C05370=1019.467,-110.317,-113.060,-23.964,21.692,-44.427
C05371=1019.463,-110.709,-113.032,-23.963,21.693,-44.433
C05372=1019.458,-111.102,-113.004,-23.963,21.694,-44.439
C05373=1019.453,-111.495,-112.976,-23.962,21.694,-44.446
C05374=1019.448,-111.888,-112.949,-23.961,21.694,-44.451
C05375=1019.443,-112.281,-112.921,-23.960,21.695,-44.456
C05376=1019.437,-112.673,-112.893,-23.959,21.696,-44.462
C05377=1019.433,-113.065,-112.866,-23.959,21.696,-44.468
C05378=1019.428,-113.458,-112.838,-23.958,21.697,-44.473
C05379=1019.423,-113.850,-112.811,-23.957,21.698,-44.479
C05380=1019.418,-114.243,-112.783,-23.957,21.699,-44.485
C05381=1019.412,-114.635,-112.756,-23.956,21.700,-44.490
C05382=1019.407,-115.028,-112.728,-23.955,21.701,-44.496
C05383=1019.402,-115.420,-112.701,-23.954,21.700,-44.501
C05384=1019.397,-115.813,-112.673,-23.954,21.701,-44.507
C05385=1019.392,-116.205,-112.645,-23.953,21.702,-44.512
C05386=1019.387,-116.598,-112.617,-23.952,21.703,-44.518
C05387=1019.381,-116.990,-112.590,-23.952,21.704,-44.523
C05388=1019.376,-117.382,-112.562,-23.951,21.705,-44.529
C05389=1019.370,-117.774,-112.535,-23.950,21.705,-44.536
C05390=1019.365,-118.167,-112.507,-23.949,21.705,-44.541
C05391=1019.360,-118.558,-112.480,-23.948,21.706,-44.547
C05392=1019.354,-118.951,-112.452,-23.948,21.706,-44.553
C05393=1019.349,-119.343,-112.425,-23.947,21.707,-44.558
C05394=1019.343,-119.736,-112.398,-23.946,21.708,-44.564
C05395=1019.338,-120.127,-112.370,-23.946,21.709,-44.569
C05396=1019.332,-120.520,-112.343,-23.945,21.710,-44.575
C05397=1019.327,-120.912,-112.315,-23.944,21.710,-44.580
C05398=1019.321,-121.304,-112.288,-23.943,21.710,-44.586
C05399=1019.315,-121.696,-112.260,-23.943,21.711,-44.591
C05400=1019.310,-122.088,-112.233,-23.942,21.712,-44.597
C05401=1019.304,-122.480,-112.206,-23.941,21.713,-44.603
C05402=1019.299,-122.872,-112.179,-23.941,21.714,-44.608
C05403=1019.292,-123.264,-112.151,-23.940,21.715,-44.614
C05404=1019.287,-123.656,-112.124,-23.939,21.714,-44.619
C05405=1019.281,-124.049,-112.097,-23.939,21.715,-44.625
C05406=1019.275,-124.440,-112.070,-23.938,21.716,-44.630
C05407=1019.269,-124.832,-112.042,-23.937,21.717,-44.636
C05408=1019.264,-125.224,-112.015,-23.936,21.718,-44.642
C05409=1019.257,-125.616,-111.988,-23.936,21.719,-44.647
C05410=1019.252,-126.008,-111.961,-23.935,21.719,-44.652
C05411=1019.246,-126.399,-111.934,-23.934,21.719,-44.658
C05412=1019.240,-126.792,-111.906,-23.934,21.720,-44.664
C05413=1019.234,-127.183,-111.880,-23.933,21.721,-44.669
C05414=1019.228,-127.576,-111.852,-23.932,21.722,-44.675
C05415=1019.222,-127.967,-111.825,-23.932,21.723,-44.680
C05416=1019.216,-128.359,-111.798,-23.931,21.723,-44.686
C05417=1019.210,-128.751,-111.771,-23.930,21.723,-44.691
C05418=1019.203,-129.143,-111.744,-23.929,21.724,-44.697
C05419=1019.198,-129.534,-111.717,-23.929,21.725,-44.703
C05420=1019.191,-129.927,-111.690,-23.928,21.726,-44.708
C05421=1019.185,-130.318,-111.663,-23.927,21.727,-44.714
C05422=1019.179,-130.711,-111.636,-23.926,21.727,-44.719
C05423=1019.173,-131.102,-111.609,-23.926,21.728,-44.725
C05424=1019.167,-131.493,-111.582,-23.925,21.728,-44.730
C05425=1019.160,-131.886,-111.555,-23.924,21.729,-44.736
C05426=1019.154,-132.277,-111.528,-23.924,21.730,-44.741
C05427=1019.148,-132.669,-111.501,-23.923,21.730,-44.747
C05428=1019.141,-133.061,-111.474,-23.922,21.731,-44.752
C05429=1019.135,-133.452,-111.448,-23.922,21.732,-44.758
C05430=1019.128,-133.844,-111.420,-23.921,21.732,-44.763
C05431=1019.504,-133.817,-111.655,-23.921,21.732,-44.763
C05432=1019.511,-133.425,-111.682,-23.922,21.732,-44.758
C05433=1019.517,-133.034,-111.709,-23.922,21.731,-44.752
C05434=1019.524,-132.641,-111.736,-23.923,21.730,-44.747
C05435=1019.530,-132.250,-111.762,-23.924,21.730,-44.741
C05436=1019.537,-131.858,-111.790,-23.924,21.729,-44.736
C05437=1019.542,-131.466,-111.816,-23.925,21.728,-44.730
C05438=1019.548,-131.075,-111.843,-23.926,21.728,-44.725
C05439=1019.554,-130.683,-111.871,-23.926,21.727,-44.719
C05440=1019.560,-130.291,-111.897,-23.927,21.727,-44.714
C05441=1019.567,-129.899,-111.924,-23.928,21.726,-44.708
C05442=1019.573,-129.508,-111.951,-23.929,21.725,-44.703
C05443=1019.578,-129.116,-111.978,-23.929,21.724,-44.697
C05444=1019.585,-128.723,-112.005,-23.930,21.723,-44.691
C05445=1019.591,-128.332,-112.032,-23.931,21.723,-44.686
C05446=1019.596,-127.940,-112.059,-23.932,21.723,-44.680
C05447=1019.603,-127.548,-112.086,-23.932,21.722,-44.675
C05448=1019.609,-127.157,-112.113,-23.933,21.721,-44.669
C05449=1019.615,-126.764,-112.141,-23.934,21.720,-44.664
C05450=1019.621,-126.373,-112.167,-23.934,21.719,-44.658
C05451=1019.626,-125.981,-112.194,-23.935,21.719,-44.652
C05452=1019.633,-125.589,-112.222,-23.936,21.719,-44.647
C05453=1019.638,-125.197,-112.249,-23.936,21.718,-44.642
C05454=1019.643,-124.805,-112.276,-23.937,21.717,-44.636
C05455=1019.650,-124.413,-112.303,-23.938,21.716,-44.630
C05456=1019.655,-124.021,-112.330,-23.939,21.715,-44.625
C05457=1019.661,-123.629,-112.357,-23.939,21.714,-44.619
C05458=1019.666,-123.237,-112.385,-23.940,21.715,-44.614
C05459=1019.672,-122.845,-112.411,-23.941,21.714,-44.608
C05460=1019.678,-122.453,-112.439,-23.941,21.713,-44.603
C05461=1019.684,-122.061,-112.466,-23.942,21.712,-44.597
C05462=1019.689,-121.669,-112.493,-23.943,21.711,-44.591
C05463=1019.695,-121.277,-112.521,-23.943,21.710,-44.586
C05464=1019.700,-120.885,-112.548,-23.944,21.710,-44.580
C05465=1019.705,-120.493,-112.576,-23.945,21.710,-44.575
C05466=1019.711,-120.101,-112.603,-23.946,21.709,-44.569
C05467=1019.716,-119.709,-112.630,-23.946,21.708,-44.564
C05468=1019.722,-119.316,-112.657,-23.947,21.707,-44.558
C05469=1019.727,-118.924,-112.684,-23.948,21.706,-44.553
C05470=1019.732,-118.532,-112.712,-23.948,21.706,-44.547
C05471=1019.738,-118.140,-112.740,-23.949,21.705,-44.541
C05472=1019.743,-117.748,-112.767,-23.950,21.705,-44.536
C05473=1019.749,-117.355,-112.795,-23.951,21.705,-44.529
C05474=1019.754,-116.963,-112.822,-23.952,21.704,-44.523
C05475=1019.759,-116.570,-112.850,-23.952,21.703,-44.518
C05476=1019.764,-116.178,-112.877,-23.953,21.702,-44.512
C05477=1019.769,-115.786,-112.904,-23.954,21.701,-44.507
C05478=1019.774,-115.393,-112.932,-23.954,21.700,-44.501
C05479=1019.779,-115.001,-112.959,-23.955,21.701,-44.496
C05480=1019.785,-114.608,-112.987,-23.956,21.700,-44.490
C05481=1019.789,-114.216,-113.014,-23.957,21.699,-44.485
C05482=1019.795,-113.823,-113.042,-23.957,21.698,-44.479
C05483=1019.800,-113.432,-113.070,-23.958,21.697,-44.473
C05484=1019.805,-113.039,-113.098,-23.959,21.696,-44.468
C05485=1019.810,-112.647,-113.125,-23.959,21.696,-44.462
C05486=1019.815,-112.254,-113.153,-23.960,21.695,-44.456
C05487=1019.819,-111.862,-113.181,-23.961,21.694,-44.451
C05488=1019.825,-111.469,-113.209,-23.962,21.694,-44.446
C05489=1019.829,-111.076,-113.236,-23.963,21.694,-44.439
C05490=1019.834,-110.683,-113.263,-23.963,21.693,-44.433
C05491=1019.839,-110.290,-113.291,-23.964,21.692,-44.427
C05492=1019.844,-109.898,-113.319,-23.965,21.691,-44.422
C05493=1019.849,-109.505,-113.347,-23.965,21.691,-44.416
C05494=1019.854,-109.112,-113.375,-23.966,21.690,-44.411
C05495=1019.858,-108.719,-113.403,-23.967,21.689,-44.405
C05496=1019.863,-108.326,-113.431,-23.968,21.688,-44.399
C05497=1019.867,-107.934,-113.459,-23.968,21.688,-44.394
C05498=1019.872,-107.541,-113.487,-23.969,21.687,-44.388
C05499=1019.877,-107.147,-113.514,-23.970,21.687,-44.383
C05500=1019.881,-106.754,-113.543,-23.971,21.686,-44.376
C05501=1019.886,-106.362,-113.570,-23.971,21.686,-44.370
C05502=1019.891,-105.969,-113.598,-23.972,21.685,-44.365
C05503=1019.895,-105.576,-113.627,-23.973,21.684,-44.359
C05504=1019.900,-105.183,-113.655,-23.974,21.683,-44.353
C05505=1019.904,-104.791,-113.682,-23.974,21.682,-44.348
C05506=1019.909,-104.399,-113.710,-23.975,21.681,-44.342
C05507=1019.913,-104.008,-113.738,-23.976,21.682,-44.337
C05508=1019.918,-103.616,-113.766,-23.976,21.681,-44.331
C05509=1019.921,-103.227,-113.794,-23.977,21.680,-44.326
C05510=1019.926,-102.836,-113.822,-23.978,21.679,-44.320
C05511=1019.930,-102.447,-113.849,-23.979,21.678,-44.314
C05512=1019.935,-102.059,-113.878,-23.980,21.678,-44.307
C05513=1019.939,-101.672,-113.905,-23.980,21.677,-44.302
C05514=1019.943,-101.284,-113.933,-23.981,21.676,-44.296
C05515=1019.947,-100.898,-113.961,-23.982,21.677,-44.291
C05516=1019.952,-100.513,-113.988,-23.982,21.676,-44.285
C05517=1019.956,-100.127,-114.016,-23.983,21.675,-44.280
C05518=1019.960,-99.743,-114.044,-23.984,21.674,-44.274
C05519=1019.964,-99.358,-114.072,-23.985,21.673,-44.268
C05520=1019.968,-98.975,-114.099,-23.985,21.673,-44.263
C05521=1019.972,-98.591,-114.127,-23.986,21.673,-44.258
C05522=1019.976,-98.208,-114.154,-23.987,21.672,-44.252
C05523=1019.980,-97.825,-114.182,-23.988,21.671,-44.246
C05524=1019.984,-97.442,-114.209,-23.988,21.670,-44.241
C05525=1019.988,-97.058,-114.238,-23.989,21.669,-44.235
C05526=1019.991,-96.675,-114.265,-23.990,21.669,-44.230
C05527=1019.996,-96.291,-114.293,-23.990,21.668,-44.224
C05528=1020.000,-95.907,-114.321,-23.991,21.668,-44.219
C05529=1020.004,-95.522,-114.348,-23.992,21.667,-44.213
C05530=1020.007,-95.138,-114.376,-23.993,21.666,-44.207
C05531=1020.011,-94.752,-114.404,-23.994,21.666,-44.200
C05532=1020.015,-94.365,-114.432,-23.994,21.665,-44.195
C05533=1020.019,-93.979,-114.461,-23.995,21.664,-44.189
C05534=1020.023,-93.592,-114.489,-23.996,21.664,-44.184
C05535=1020.026,-93.203,-114.516,-23.996,21.664,-44.178
C05536=1020.027,-93.059,-114.527,-23.997,21.663,-44.176
C05537=1019.643,111.857,-131.928,-24.335,21.425,-41.686
C05538=1019.639,112.243,-131.965,-24.335,21.423,-41.684
C05539=1019.635,112.628,-132.001,-24.335,21.424,-41.681
C05540=1019.630,113.026,-132.039,-24.336,21.423,-41.677
C05541=1019.625,113.425,-132.077,-24.336,21.423,-41.675
C05542=1019.620,113.823,-132.115,-24.337,21.423,-41.671
C05543=1019.616,114.222,-132.152,-24.337,21.422,-41.668
C05544=1019.611,114.620,-132.190,-24.338,21.423,-41.664
C05545=1019.606,115.019,-132.228,-24.338,21.422,-41.662
C05546=1019.602,115.418,-132.266,-24.339,21.422,-41.659
C05547=1019.597,115.816,-132.304,-24.339,21.422,-41.655
C05548=1019.592,116.214,-132.341,-24.340,21.422,-41.652
C05549=1019.588,116.613,-132.380,-24.340,21.421,-41.649
C05550=1019.583,117.012,-132.417,-24.340,21.420,-41.646
C05551=1019.578,117.410,-132.455,-24.341,21.421,-41.642
C05552=1019.573,117.809,-132.493,-24.341,21.420,-41.638
C05553=1019.568,118.207,-132.531,-24.342,21.420,-41.637
C05554=1019.563,118.606,-132.569,-24.342,21.420,-41.633
C05555=1019.559,119.004,-132.607,-24.343,21.420,-41.629
C05556=1019.553,119.403,-132.644,-24.343,21.420,-41.626
C05557=1019.549,119.801,-132.683,-24.343,21.419,-41.624
C05558=1019.544,120.200,-132.721,-24.344,21.419,-41.620
C05559=1019.539,120.599,-132.759,-24.345,21.419,-41.617
C05560=1019.534,120.997,-132.797,-24.345,21.418,-41.614
C05561=1019.530,121.395,-132.835,-24.345,21.418,-41.611
C05562=1019.525,121.794,-132.873,-24.346,21.418,-41.607
C05563=1019.521,122.192,-132.912,-24.346,21.417,-41.605
C05564=1019.516,122.591,-132.949,-24.347,21.418,-41.602
C05565=1019.511,122.990,-132.988,-24.347,21.417,-41.598
C05566=1019.507,123.388,-133.026,-24.348,21.418,-41.595
C05567=1019.502,123.787,-133.064,-24.348,21.416,-41.592
C05568=1019.498,124.185,-133.103,-24.348,21.417,-41.589
C05569=1019.492,124.584,-133.140,-24.349,21.416,-41.585
C05570=1019.488,124.982,-133.179,-24.349,21.416,-41.583
C05571=1019.483,125.381,-133.217,-24.350,21.416,-41.580
C05572=1019.479,125.779,-133.255,-24.350,21.416,-41.576
C05573=1019.474,126.178,-133.294,-24.350,21.415,-41.574
C05574=1019.469,126.577,-133.332,-24.351,21.415,-41.571
C05575=1019.464,126.976,-133.370,-24.351,21.415,-41.567
C05576=1019.459,127.374,-133.409,-24.352,21.415,-41.565
C05577=1019.454,127.772,-133.447,-24.352,21.414,-41.561
C05578=1019.450,128.171,-133.485,-24.353,21.415,-41.558
C05579=1019.444,128.570,-133.523,-24.353,21.414,-41.555
C05580=1019.440,128.969,-133.562,-24.354,21.414,-41.552
C05581=1019.435,129.367,-133.600,-24.354,21.413,-41.550
C05582=1019.431,129.766,-133.638,-24.354,21.413,-41.547
C05583=1019.425,130.164,-133.677,-24.355,21.413,-41.543
C05584=1019.421,130.564,-133.715,-24.355,21.413,-41.541
C05585=1019.415,130.961,-133.753,-24.356,21.413,-41.538
C05586=1019.410,131.360,-133.792,-24.356,21.413,-41.534
C05587=1019.406,131.759,-133.830,-24.356,21.412,-41.532
C05588=1019.400,132.158,-133.869,-24.357,21.412,-41.528
C05589=1019.396,132.557,-133.907,-24.357,21.412,-41.525
C05590=1019.390,132.956,-133.946,-24.358,21.411,-41.523
C05591=1019.386,133.354,-133.984,-24.358,21.412,-41.519
C05592=1019.380,133.752,-134.023,-24.358,21.411,-41.517
C05593=1019.375,134.151,-134.061,-24.359,21.411,-41.514
C05594=1019.370,134.550,-134.100,-24.359,21.411,-41.510
C05595=1019.365,134.949,-134.138,-24.360,21.410,-41.508
C05596=1019.360,135.347,-134.177,-24.360,21.411,-41.505
C05597=1019.355,135.743,-134.214,-24.360,21.410,-41.502
C05598=1019.350,136.115,-134.250,-24.361,21.409,-41.500
C05599=1019.346,136.454,-134.283,-24.361,21.410,-41.497
C05600=1019.342,136.772,-134.314,-24.361,21.409,-41.495
C05601=1019.338,137.088,-134.345,-24.362,21.409,-41.491
C05602=1019.334,137.424,-134.377,-24.363,21.410,-41.488
C05603=1019.329,137.794,-134.413,-24.363,21.408,-41.486
C05604=1019.323,138.196,-134.452,-24.363,21.408,-41.484
C05605=1019.320,138.402,-134.471,-24.363,21.408,-41.482
C05606=1019.317,138.618,-134.492,-24.364,21.408,-41.480
C05607=1019.315,138.855,-134.515,-24.364,21.408,-41.478
C05608=1019.311,139.115,-134.541,-24.364,21.407,-41.476
C05609=1019.307,139.393,-134.567,-24.364,21.408,-41.475
C05610=1019.304,139.681,-134.596,-24.365,21.408,-41.473
C05611=1019.300,139.969,-134.623,-24.365,21.408,-41.471
C05612=1019.296,140.246,-134.650,-24.365,21.408,-41.470
C05613=1019.293,140.504,-134.675,-24.366,21.408,-41.468
C05614=1019.290,140.740,-134.697,-24.366,21.408,-41.466
C05615=1019.284,141.158,-134.738,-24.366,21.407,-41.462
C05616=1019.279,141.562,-134.777,-24.366,21.406,-41.460
C05617=1019.273,141.968,-134.817,-24.367,21.407,-41.457
C05618=1019.268,142.374,-134.855,-24.368,21.406,-41.453
C05619=1019.263,142.781,-134.895,-24.368,21.406,-41.451
C05620=1019.257,143.189,-134.935,-24.368,21.406,-41.448
C05621=1019.252,143.598,-134.974,-24.369,21.405,-41.445
C05622=1019.246,144.007,-135.014,-24.369,21.406,-41.442
C05623=1019.240,144.418,-135.054,-24.370,21.405,-41.438
C05624=1019.235,144.828,-135.093,-24.370,21.405,-41.436
C05625=1019.229,145.241,-135.133,-24.370,21.405,-41.432
C05626=1019.224,145.652,-135.173,-24.371,21.404,-41.431
C05627=1019.218,146.065,-135.214,-24.371,21.405,-41.427
C05628=1019.212,146.477,-135.254,-24.372,21.404,-41.424
C05629=1019.207,146.891,-135.293,-24.372,21.404,-41.422
C05630=1019.201,147.304,-135.334,-24.372,21.404,-41.418
C05631=1019.195,147.718,-135.374,-24.373,21.403,-41.416
C05632=1019.189,148.133,-135.414,-24.373,21.403,-41.412
C05633=1019.183,148.546,-135.455,-24.374,21.403,-41.409
C05634=1019.178,148.960,-135.495,-24.374,21.403,-41.407
C05635=1019.172,149.375,-135.535,-24.375,21.403,-41.403
C05636=1019.166,149.789,-135.575,-24.375,21.402,-41.401
C05637=1019.161,150.203,-135.615,-24.375,21.402,-41.398
C05638=1019.155,150.617,-135.655,-24.376,21.402,-41.394
C05639=1019.149,151.030,-135.695,-24.376,21.401,-41.392
C05640=1019.143,151.444,-135.736,-24.377,21.402,-41.389
C05641=1019.137,151.857,-135.776,-24.377,21.402,-41.387
C05642=1019.131,152.271,-135.816,-24.377,21.401,-41.383
C05643=1019.125,152.683,-135.856,-24.378,21.401,-41.381
C05644=1019.118,153.096,-135.896,-24.378,21.400,-41.377
C05645=1019.113,153.507,-135.936,-24.378,21.400,-41.375
C05646=1019.107,153.918,-135.977,-24.379,21.401,-41.372
C05647=1019.101,154.329,-136.017,-24.380,21.400,-41.368
C05648=1019.095,154.739,-136.056,-24.380,21.400,-41.366
C05649=1019.089,155.149,-136.096,-24.380,21.400,-41.363
C05650=1019.083,155.557,-136.136,-24.381,21.399,-41.361
C05651=1019.077,155.965,-136.176,-24.381,21.400,-41.358
C05652=1019.071,156.371,-136.215,-24.381,21.399,-41.355
C05653=1019.065,156.777,-136.255,-24.382,21.399,-41.352
C05654=1019.059,157.182,-136.294,-24.382,21.399,-41.350
C05655=1019.053,157.587,-136.334,-24.383,21.398,-41.346
C05656=1019.047,157.990,-136.373,-24.383,21.398,-41.344
C05657=1019.041,158.392,-136.413,-24.383,21.399,-41.341
C05658=1019.036,158.794,-136.452,-24.384,21.397,-41.339
C05659=1019.029,159.196,-136.491,-24.384,21.398,-41.335
C05660=1019.024,159.597,-136.530,-24.384,21.398,-41.333
C05661=1019.023,159.997,-136.573,-24.385,21.397,-41.330
C05662=1019.021,160.393,-136.614,-24.385,21.397,-41.328
C05663=1019.020,160.798,-136.656,-24.386,21.397,-41.325
C05664=1019.020,161.012,-136.679,-24.386,21.397,-41.324
C05665=1019.018,161.237,-136.702,-24.386,21.396,-41.322
C05666=1019.018,161.474,-136.727,-24.386,21.396,-41.320
C05667=1019.016,161.725,-136.753,-24.387,21.397,-41.319
C05668=1019.016,161.988,-136.781,-24.387,21.397,-41.317
C05669=1019.015,162.256,-136.809,-24.387,21.396,-41.315
C05670=1019.015,162.529,-136.837,-24.387,21.396,-41.313
C05671=1019.013,162.797,-136.866,-24.388,21.396,-41.311
C05672=1019.012,163.060,-136.893,-24.388,21.396,-41.309
C05673=1019.011,163.314,-136.920,-24.388,21.395,-41.308
C05674=1019.011,163.549,-136.945,-24.388,21.396,-41.306
C05675=1019.010,163.961,-136.989,-24.389,21.395,-41.304
C05676=1019.009,164.152,-137.008,-24.389,21.395,-41.302
C05677=1019.008,164.537,-137.049,-24.389,21.395,-41.300
C05678=1019.006,164.937,-137.091,-24.390,21.395,-41.297
C05679=1019.005,165.338,-137.133,-24.390,21.395,-41.295
C05680=1019.004,165.738,-137.176,-24.390,21.394,-41.291
C05681=1019.002,166.139,-137.217,-24.391,21.394,-41.289
C05682=1019.002,166.539,-137.259,-24.391,21.395,-41.286
C05683=1019.000,166.940,-137.302,-24.391,21.393,-41.284
C05684=1018.999,167.339,-137.344,-24.392,21.394,-41.280
C05685=1018.997,167.740,-137.387,-24.392,21.394,-41.278
C05686=1018.996,168.141,-137.428,-24.393,21.394,-41.275
C05687=1018.995,168.541,-137.471,-24.393,21.393,-41.273
C05688=1018.993,168.942,-137.513,-24.393,21.393,-41.271
C05689=1018.992,169.342,-137.555,-24.394,21.393,-41.267
C05690=1018.991,169.742,-137.598,-24.394,21.392,-41.265
C05691=1018.990,170.143,-137.640,-24.395,21.392,-41.262
C05692=1018.989,170.544,-137.683,-24.395,21.392,-41.260
C05693=1018.987,170.944,-137.726,-24.395,21.392,-41.256
C05694=1018.986,171.345,-137.768,-24.396,21.392,-41.254
C05695=1018.985,171.745,-137.811,-24.396,21.392,-41.251
C05696=1018.984,172.146,-137.853,-24.396,21.392,-41.249
C05697=1018.983,172.547,-137.895,-24.397,21.391,-41.247
C05698=1018.981,172.947,-137.938,-24.397,21.391,-41.243
C05699=1018.981,173.347,-137.980,-24.397,21.391,-41.242
C05700=1018.979,173.749,-138.023,-24.398,21.390,-41.238
C05701=1018.978,174.149,-138.066,-24.398,21.390,-41.236
C05702=1018.976,174.550,-138.109,-24.399,21.391,-41.233
C05703=1018.975,174.950,-138.150,-24.399,21.390,-41.231
C05704=1018.975,175.352,-138.193,-24.400,21.390,-41.227
C05705=1018.973,175.752,-138.236,-24.400,21.390,-41.225
C05706=1018.972,176.153,-138.279,-24.400,21.390,-41.223
C05707=1018.971,176.553,-138.321,-24.401,21.389,-41.219
C05708=1018.970,176.954,-138.364,-24.401,21.389,-41.218
C05709=1018.969,177.355,-138.407,-24.401,21.389,-41.214
C05710=1018.968,177.756,-138.450,-24.402,21.389,-41.212
C05711=1018.966,178.156,-138.493,-24.402,21.389,-41.209
C05712=1018.966,178.558,-138.535,-24.402,21.388,-41.207
C05713=1018.965,178.958,-138.578,-24.403,21.388,-41.205
C05714=1018.963,179.359,-138.621,-24.403,21.388,-41.201
C05715=1018.963,179.760,-138.664,-24.403,21.388,-41.199
C05716=1018.961,180.160,-138.707,-24.404,21.388,-41.196
C05717=1018.960,180.562,-138.751,-24.404,21.388,-41.194
C05718=1018.959,180.963,-138.793,-24.405,21.387,-41.190
C05719=1018.957,181.363,-138.836,-24.405,21.387,-41.188
C05720=1018.957,181.764,-138.879,-24.405,21.387,-41.186
C05721=1018.957,182.165,-138.922,-24.406,21.387,-41.183
C05722=1018.955,182.566,-138.965,-24.406,21.386,-41.181
C05723=1018.955,182.967,-139.008,-24.407,21.387,-41.177
C05724=1018.953,183.368,-139.051,-24.407,21.386,-41.176
C05725=1018.952,183.769,-139.094,-24.407,21.386,-41.172
C05726=1018.951,184.169,-139.137,-24.408,21.386,-41.170
C05727=1018.950,184.571,-139.181,-24.408,21.386,-41.168
C05728=1018.950,184.972,-139.224,-24.409,21.386,-41.165
C05729=1018.948,185.372,-139.267,-24.409,21.385,-41.162
C05730=1018.948,185.773,-139.310,-24.409,21.385,-41.159
C05731=1018.947,186.175,-139.354,-24.410,21.385,-41.157
C05732=1018.945,186.575,-139.397,-24.410,21.384,-41.155
C05733=1018.945,186.976,-139.440,-24.410,21.384,-41.151
C05734=1018.944,187.378,-139.483,-24.411,21.384,-41.150
C05735=1018.943,187.779,-139.526,-24.411,21.385,-41.146
C05736=1018.942,188.179,-139.569,-24.411,21.384,-41.144
C05737=1018.941,188.581,-139.613,-24.412,21.384,-41.141
C05738=1018.940,188.982,-139.656,-24.412,21.384,-41.139
C05739=1018.940,189.383,-139.699,-24.412,21.384,-41.137
C05740=1018.939,189.784,-139.743,-24.413,21.383,-41.133
C05741=1018.938,190.185,-139.787,-24.413,21.383,-41.131
C05742=1018.937,190.586,-139.831,-24.414,21.383,-41.128
C05743=1018.936,190.988,-139.874,-24.414,21.383,-41.126
C05744=1018.935,191.389,-139.917,-24.414,21.382,-41.124
C05745=1018.935,191.790,-139.961,-24.415,21.382,-41.120
C05746=1018.934,192.191,-140.005,-24.415,21.382,-41.118
C05747=1018.933,192.592,-140.048,-24.415,21.382,-41.115
C05748=1018.932,192.992,-140.091,-24.416,21.382,-41.113
C05749=1018.931,193.395,-140.135,-24.416,21.382,-41.109
C05750=1018.931,193.795,-140.179,-24.417,21.382,-41.108
C05751=1018.930,194.196,-140.222,-24.417,21.381,-41.105
C05752=1018.929,194.598,-140.266,-24.417,21.381,-41.102
C05753=1018.929,194.998,-140.310,-24.418,21.381,-41.100
C05754=1018.928,195.399,-140.353,-24.418,21.381,-41.097
C05755=1018.927,195.801,-140.397,-24.418,21.380,-41.094
C05756=1018.926,196.201,-140.441,-24.419,21.381,-41.091
C05757=1018.926,196.603,-140.485,-24.419,21.380,-41.089
C05758=1018.926,197.004,-140.529,-24.419,21.380,-41.087
C05759=1018.925,197.405,-140.572,-24.420,21.380,-41.084
C05760=1018.923,197.807,-140.616,-24.420,21.380,-41.082
C05761=1018.923,198.207,-140.660,-24.421,21.380,-41.078
C05762=1018.923,198.609,-140.704,-24.421,21.379,-41.076
C05763=1018.922,199.010,-140.748,-24.421,21.379,-41.074
C05764=1018.922,199.408,-140.791,-24.422,21.379,-41.071
C05765=1018.921,199.797,-140.834,-24.422,21.379,-41.069
C05766=1018.920,200.198,-140.878,-24.423,21.378,-41.065
C05767=1018.920,200.411,-140.901,-24.423,21.378,-41.065
C05768=1018.920,200.633,-140.926,-24.423,21.378,-41.063
C05769=1018.920,200.863,-140.951,-24.423,21.378,-41.061
C05770=1018.919,201.090,-140.976,-24.423,21.379,-41.060
C05771=1018.919,201.497,-141.020,-24.424,21.378,-41.058
C05772=1018.919,201.848,-141.059,-24.424,21.378,-41.054
C05773=1018.920,202.198,-141.099,-24.424,21.378,-41.052
C05774=1018.920,202.585,-141.142,-24.425,21.378,-41.051
C05775=1018.927,203.801,-141.279,-24.373,21.403,-41.416
C05776=1018.929,204.050,-141.306,-24.373,21.404,-41.415
C05777=1018.931,204.298,-141.333,-24.373,21.403,-41.414
C05778=1018.933,204.546,-141.361,-24.373,21.403,-41.412
C05779=1018.935,204.795,-141.388,-24.374,21.404,-41.411
C05780=1018.937,205.043,-141.415,-24.373,21.403,-41.410
C05781=1018.939,205.292,-141.443,-24.374,21.403,-41.409
C05782=1018.941,205.540,-141.470,-24.374,21.403,-41.407
C05783=1018.943,205.790,-141.498,-24.374,21.402,-41.407
C05784=1018.945,206.038,-141.526,-24.374,21.403,-41.405
C05785=1018.947,206.286,-141.553,-24.375,21.403,-41.403
C05786=1018.949,206.556,-141.583,-24.375,21.402,-41.401
C05787=1018.951,206.826,-141.613,-24.375,21.402,-41.401
C05788=1018.954,207.097,-141.643,-24.375,21.402,-41.399
C05789=1018.956,207.367,-141.672,-24.375,21.402,-41.398
C05790=1018.957,207.615,-141.701,-24.376,21.403,-41.396
C05791=1018.959,207.863,-141.728,-24.376,21.402,-41.396
C05792=1018.962,208.113,-141.755,-24.376,21.402,-41.394
C05793=1018.964,208.361,-141.783,-24.376,21.402,-41.392
C05794=1018.965,208.593,-141.808,-24.376,21.402,-41.391
C05795=1018.967,208.824,-141.835,-24.376,21.401,-41.390
C05796=1018.969,209.057,-141.860,-24.377,21.402,-41.389
C05797=1018.971,209.288,-141.886,-24.377,21.402,-41.387
C05798=1018.974,209.520,-141.912,-24.377,21.402,-41.387
C05799=1018.975,209.751,-141.937,-24.377,21.401,-41.385
C05800=1018.977,209.983,-141.963,-24.377,21.401,-41.383
C05801=1018.979,210.216,-141.989,-24.377,21.401,-41.383
C05802=1018.981,210.464,-142.017,-24.378,21.401,-41.381
C05803=1018.983,210.712,-142.044,-24.378,21.401,-41.379
C05804=1018.985,210.960,-142.072,-24.378,21.401,-41.378
C05805=1018.987,211.209,-142.099,-24.378,21.400,-41.377
C05806=1018.990,211.458,-142.127,-24.378,21.400,-41.375
C05807=1018.991,211.706,-142.156,-24.379,21.401,-41.374
C05808=1018.993,211.954,-142.183,-24.379,21.401,-41.372
C05809=1018.996,212.203,-142.211,-24.379,21.400,-41.372
C05810=1018.998,212.452,-142.238,-24.379,21.400,-41.370
C05811=1019.000,212.700,-142.266,-24.380,21.400,-41.368
C05812=1019.002,212.948,-142.293,-24.380,21.400,-41.366
C05813=1019.004,213.197,-142.322,-24.380,21.400,-41.366
C05814=1019.007,213.445,-142.349,-24.380,21.400,-41.365
C05815=1019.008,213.694,-142.377,-24.380,21.400,-41.363
C05816=1019.011,213.942,-142.405,-24.381,21.400,-41.361
C05817=1019.013,214.190,-142.433,-24.381,21.400,-41.359
C05818=1019.015,214.439,-142.460,-24.381,21.399,-41.359
C05819=1019.018,214.688,-142.488,-24.381,21.399,-41.357
C05820=1019.020,214.935,-142.516,-24.381,21.400,-41.356
C05821=1019.021,215.184,-142.544,-24.382,21.399,-41.354
C05822=1019.024,215.427,-142.571,-24.382,21.398,-41.353
C05823=1019.027,215.670,-142.598,-24.382,21.399,-41.352
C05824=1019.029,215.913,-142.626,-24.382,21.399,-41.350
C05825=1019.031,216.155,-142.653,-24.382,21.399,-41.348
C05826=1019.033,216.399,-142.680,-24.383,21.398,-41.346
C05827=1019.035,216.641,-142.707,-24.383,21.398,-41.346
C05828=1019.037,216.884,-142.734,-24.383,21.398,-41.344
C05829=1019.040,217.126,-142.761,-24.383,21.398,-41.342
C05830=1019.042,217.375,-142.790,-24.383,21.399,-41.341
C05831=1019.044,217.624,-142.817,-24.384,21.398,-41.339
C05832=1019.046,217.872,-142.845,-24.384,21.397,-41.339
C05833=1019.049,218.120,-142.873,-24.384,21.397,-41.337
C05834=1019.051,218.368,-142.901,-24.384,21.398,-41.335
C05835=1019.053,218.617,-142.930,-24.384,21.398,-41.333
C05836=1019.055,218.866,-142.957,-24.385,21.397,-41.332
C05837=1019.058,219.114,-142.985,-24.385,21.397,-41.330
C05838=1019.060,219.362,-143.013,-24.385,21.397,-41.330
C05839=1019.063,219.611,-143.041,-24.385,21.397,-41.328
C05840=1019.065,219.859,-143.069,-24.385,21.397,-41.326
C05841=1019.067,220.108,-143.097,-24.386,21.397,-41.324
C05842=1019.070,220.356,-143.125,-24.386,21.397,-41.323
C05843=1019.073,220.604,-143.153,-24.386,21.397,-41.321
C05844=1019.074,220.853,-143.181,-24.386,21.396,-41.320
C05845=1019.077,221.102,-143.209,-24.386,21.396,-41.318
C05846=1019.079,221.350,-143.237,-24.387,21.397,-41.317
C05847=1019.082,221.598,-143.265,-24.387,21.396,-41.315
C05848=1019.084,221.846,-143.293,-24.387,21.396,-41.313
C05849=1019.087,222.095,-143.321,-24.388,21.396,-41.311
C05850=1019.088,222.338,-143.349,-24.388,21.397,-41.310
C05851=1019.091,222.581,-143.376,-24.388,21.396,-41.309
C05852=1019.094,222.824,-143.404,-24.388,21.395,-41.308
C05853=1019.095,223.066,-143.431,-24.388,21.395,-41.306
C05854=1019.098,223.310,-143.459,-24.389,21.396,-41.304
C05855=1019.101,223.552,-143.486,-24.389,21.396,-41.302
C05856=1019.104,223.795,-143.514,-24.389,21.395,-41.300
C05857=1019.105,224.038,-143.541,-24.389,21.395,-41.300
C05858=1019.108,224.287,-143.569,-24.389,21.394,-41.298
C05859=1019.111,224.535,-143.597,-24.390,21.395,-41.297
C05860=1019.113,224.784,-143.626,-24.390,21.395,-41.295
C05861=1019.116,225.032,-143.655,-24.390,21.395,-41.293
C05862=1019.118,225.279,-143.682,-24.390,21.394,-41.291
C05863=1019.121,225.528,-143.711,-24.391,21.394,-41.289
C05864=1019.124,225.777,-143.739,-24.391,21.395,-41.288
C05865=1019.125,226.025,-143.767,-24.391,21.395,-41.286
C05866=1019.128,226.274,-143.795,-24.391,21.394,-41.285
C05867=1019.131,226.522,-143.823,-24.391,21.393,-41.284
C05868=1019.133,226.771,-143.852,-24.392,21.393,-41.282
C05869=1019.136,227.018,-143.881,-24.392,21.394,-41.280
C05870=1019.139,227.267,-143.909,-24.392,21.394,-41.278
C05871=1019.141,227.515,-143.937,-24.393,21.393,-41.276
C05872=1019.144,227.764,-143.965,-24.393,21.393,-41.275
C05873=1019.147,228.012,-143.993,-24.393,21.393,-41.273
C05874=1019.148,228.261,-144.021,-24.393,21.394,-41.271
C05875=1019.151,228.509,-144.050,-24.394,21.393,-41.269
C05876=1019.154,228.757,-144.078,-24.394,21.393,-41.267
C05877=1019.157,229.006,-144.107,-24.394,21.393,-41.266
C05878=1019.159,229.249,-144.134,-24.394,21.392,-41.265
C05879=1019.162,229.491,-144.162,-24.394,21.392,-41.263
C05880=1019.164,229.735,-144.190,-24.395,21.392,-41.262
C05881=1019.167,229.978,-144.218,-24.395,21.392,-41.260
C05882=1019.169,230.221,-144.246,-24.395,21.392,-41.258
C05883=1019.172,230.464,-144.273,-24.395,21.392,-41.256
C05884=1019.175,230.707,-144.302,-24.396,21.392,-41.254
C05885=1019.177,230.950,-144.329,-24.396,21.391,-41.252
C05886=1019.180,231.198,-144.357,-24.396,21.392,-41.251
C05887=1019.183,231.447,-144.386,-24.396,21.392,-41.249
C05888=1019.185,231.695,-144.415,-24.397,21.392,-41.247
C05889=1019.188,231.944,-144.443,-24.397,21.391,-41.245
C05890=1019.192,232.192,-144.472,-24.397,21.391,-41.243
C05891=1019.193,232.440,-144.500,-24.397,21.391,-41.242
C05892=1019.196,232.688,-144.528,-24.398,21.391,-41.240
C05893=1019.199,232.936,-144.557,-24.398,21.390,-41.238
C05894=1019.202,233.185,-144.586,-24.398,21.391,-41.236
C05895=1019.205,233.433,-144.614,-24.399,21.391,-41.234
C05896=1019.207,233.682,-144.643,-24.399,21.391,-41.233
C05897=1019.210,233.931,-144.671,-24.399,21.390,-41.231
C05898=1019.213,234.178,-144.699,-24.399,21.390,-41.229
C05899=1019.215,234.427,-144.728,-24.400,21.390,-41.227
C05900=1019.218,234.675,-144.757,-24.400,21.390,-41.225
C05901=1019.221,234.923,-144.785,-24.400,21.390,-41.223
C05902=1019.224,235.172,-144.814,-24.400,21.389,-41.221
C05903=1019.227,235.420,-144.843,-24.401,21.389,-41.219
C05904=1019.230,235.668,-144.871,-24.401,21.389,-41.218
C05905=1019.232,235.917,-144.901,-24.401,21.390,-41.216
C05906=1019.235,236.160,-144.928,-24.401,21.389,-41.214
C05907=1019.238,236.403,-144.956,-24.402,21.389,-41.212
C05908=1019.241,236.646,-144.985,-24.402,21.389,-41.210
C05909=1019.243,236.889,-145.013,-24.402,21.389,-41.209
C05910=1019.246,237.132,-145.041,-24.402,21.388,-41.207
C05911=1019.249,237.375,-145.069,-24.403,21.388,-41.205
C05912=1019.252,237.619,-145.097,-24.403,21.388,-41.203
C05913=1019.255,237.861,-145.125,-24.403,21.388,-41.201
C05914=1019.257,238.110,-145.154,-24.403,21.388,-41.199
C05915=1019.260,238.358,-145.182,-24.404,21.387,-41.197
C05916=1019.264,238.606,-145.211,-24.404,21.387,-41.195
C05917=1019.266,238.855,-145.240,-24.405,21.388,-41.192
C05918=1019.269,239.103,-145.269,-24.405,21.387,-41.190
C05919=1019.272,239.351,-145.297,-24.405,21.387,-41.188
C05920=1019.275,239.599,-145.327,-24.405,21.387,-41.186
C05921=1019.278,239.849,-145.355,-24.406,21.387,-41.184
C05922=1019.281,240.097,-145.385,-24.406,21.386,-41.183
C05923=1019.284,240.345,-145.413,-24.406,21.386,-41.181
C05924=1019.288,240.593,-145.442,-24.406,21.386,-41.179
C05925=1019.290,240.842,-145.471,-24.407,21.386,-41.177
C05926=1019.293,241.090,-145.500,-24.407,21.386,-41.174
C05927=1019.296,241.338,-145.528,-24.407,21.386,-41.172
C05928=1019.299,241.586,-145.558,-24.408,21.386,-41.170
C05929=1019.302,241.835,-145.586,-24.408,21.386,-41.168
C05930=1019.305,242.084,-145.616,-24.408,21.385,-41.166
C05931=1019.308,242.332,-145.644,-24.408,21.385,-41.164
C05932=1019.311,242.580,-145.673,-24.409,21.385,-41.162
C05933=1019.314,242.828,-145.702,-24.409,21.385,-41.159
C05934=1019.317,243.071,-145.730,-24.410,21.385,-41.157
C05935=1019.320,243.315,-145.759,-24.410,21.385,-41.155
C05936=1019.323,243.557,-145.788,-24.410,21.385,-41.153
C05937=1019.326,243.801,-145.816,-24.410,21.384,-41.151
C05938=1019.329,244.044,-145.844,-24.411,21.384,-41.150
C05939=1019.332,244.287,-145.873,-24.411,21.384,-41.148
C05940=1019.335,244.530,-145.901,-24.411,21.384,-41.144
C05941=1019.338,244.774,-145.930,-24.412,21.384,-41.143
C05942=1019.341,245.022,-145.959,-24.412,21.384,-41.141
C05943=1019.344,245.270,-145.988,-24.412,21.384,-41.139
C05944=1019.348,245.519,-146.017,-24.412,21.384,-41.137
C05945=1019.351,245.767,-146.046,-24.413,21.384,-41.134
C05946=1019.353,246.015,-146.075,-24.413,21.384,-41.132
C05947=1019.357,246.263,-146.104,-24.413,21.383,-41.129
C05948=1019.360,246.512,-146.134,-24.414,21.382,-41.127
C05949=1019.363,246.760,-146.163,-24.414,21.382,-41.126
C05950=1019.366,247.008,-146.192,-24.414,21.383,-41.122
C05951=1019.369,247.256,-146.221,-24.415,21.382,-41.120
C05952=1019.373,247.505,-146.250,-24.415,21.382,-41.118
C05953=1019.375,247.753,-146.279,-24.415,21.382,-41.117
C05954=1019.379,248.002,-146.309,-24.416,21.382,-41.113
C05955=1019.382,248.250,-146.339,-24.416,21.382,-41.111
C05956=1019.385,248.498,-146.367,-24.416,21.381,-41.109
C05957=1019.389,248.746,-146.397,-24.417,21.381,-41.107
C05958=1019.392,248.995,-146.426,-24.417,21.381,-41.104
C05959=1019.395,249.242,-146.455,-24.417,21.381,-41.102
C05960=1019.398,249.491,-146.485,-24.418,21.381,-41.100
C05961=1019.401,249.739,-146.513,-24.418,21.381,-41.098
C05962=1019.404,249.983,-146.543,-24.418,21.381,-41.095
C05963=1019.408,250.226,-146.571,-24.419,21.381,-41.093
C05964=1019.411,250.469,-146.600,-24.419,21.380,-41.091
C05965=1019.415,250.713,-146.629,-24.419,21.380,-41.089
C05966=1019.418,250.956,-146.658,-24.420,21.380,-41.085
C05967=1019.420,251.199,-146.687,-24.420,21.380,-41.084
C05968=1019.424,251.443,-146.715,-24.420,21.380,-41.082
C05969=1019.427,251.686,-146.745,-24.421,21.380,-41.078
C05970=1019.431,251.934,-146.773,-24.421,21.380,-41.076
C05971=1019.434,252.183,-146.803,-24.421,21.379,-41.074
C05972=1019.437,252.431,-146.832,-24.421,21.378,-41.072
C05973=1019.440,252.679,-146.862,-24.422,21.379,-41.069
C05974=1019.444,252.927,-146.891,-24.422,21.379,-41.067
C05975=1019.448,253.175,-146.921,-24.423,21.378,-41.065
C05976=1019.450,253.424,-146.950,-24.423,21.378,-41.061
C05977=1019.454,253.672,-146.980,-24.423,21.378,-41.060
C05978=1019.457,253.920,-147.010,-24.424,21.378,-41.058
C05979=1019.461,254.169,-147.039,-24.424,21.378,-41.054
C05980=1019.464,254.416,-147.069,-24.424,21.378,-41.052
C05981=1019.468,254.665,-147.098,-24.425,21.377,-41.049
C05982=1019.470,254.913,-147.127,-24.425,21.377,-41.047
C05983=1019.474,255.161,-147.157,-24.425,21.377,-41.045
C05984=1019.477,255.410,-147.187,-24.426,21.377,-41.042
C05985=1019.481,255.658,-147.217,-24.426,21.377,-41.040
C05986=1019.485,255.906,-147.246,-24.426,21.376,-41.037
C05987=1019.488,256.154,-147.276,-24.427,21.376,-41.034
C05988=1019.492,256.402,-147.306,-24.427,21.376,-41.032
C05989=1019.494,256.650,-147.335,-24.428,21.377,-41.029
C05990=1019.498,256.894,-147.364,-24.428,21.376,-41.027
C05991=1019.501,257.137,-147.393,-24.428,21.375,-41.025
C05992=1019.505,257.381,-147.422,-24.429,21.376,-41.021
C05993=1019.508,257.625,-147.451,-24.429,21.376,-41.019
C05994=1019.513,257.868,-147.481,-24.429,21.375,-41.018
C05995=1019.516,258.112,-147.510,-24.430,21.375,-41.014
C05996=1019.519,258.355,-147.540,-24.430,21.375,-41.012
C05997=1019.537,259.591,-147.693,-24.551,21.322,-40.171
C05998=1019.539,259.870,-147.730,-24.587,21.310,-39.930
C05999=1019.542,260.150,-147.767,-24.622,21.297,-39.689
C06000=1019.543,260.430,-147.805,-24.658,21.287,-39.446
C06001=1019.545,260.710,-147.844,-24.693,21.275,-39.204
C06002=1019.546,260.957,-147.878,-24.725,21.267,-38.988
C06003=1019.546,261.204,-147.913,-24.758,21.259,-38.770
C06004=1019.546,261.452,-147.949,-24.790,21.251,-38.554
C06005=1019.546,261.700,-147.985,-24.823,21.245,-38.337
C06006=1019.546,261.979,-148.027,-24.860,21.238,-38.090
C06007=1019.545,262.259,-148.069,-24.897,21.233,-37.842
C06008=1019.543,262.538,-148.111,-24.935,21.227,-37.593
C06009=1019.541,262.817,-148.154,-24.973,21.223,-37.345
C06010=1019.539,263.063,-148.194,-25.006,21.220,-37.124
C06011=1019.537,263.311,-148.233,-25.040,21.218,-36.903
C06012=1019.534,263.558,-148.273,-25.074,21.217,-36.681
C06013=1019.530,263.804,-148.314,-25.108,21.216,-36.459
C06014=1019.526,264.083,-148.360,-25.147,21.215,-36.207
C06015=1019.522,264.363,-148.407,-25.186,21.217,-35.952
C06016=1019.517,264.642,-148.455,-25.226,21.219,-35.699
C06017=1019.511,264.921,-148.503,-25.265,21.221,-35.444
C06018=1019.505,265.167,-148.547,-25.300,21.225,-35.219
C06019=1019.500,265.414,-148.591,-25.335,21.229,-34.991
C06020=1019.494,265.659,-148.635,-25.370,21.233,-34.766
C06021=1019.488,265.905,-148.680,-25.406,21.239,-34.538
C06022=1019.480,266.184,-148.731,-25.446,21.246,-34.279
C06023=1019.472,266.463,-148.783,-25.487,21.254,-34.021
C06024=1019.464,266.742,-148.836,-25.527,21.264,-33.760
C06025=1019.455,267.020,-148.889,-25.568,21.275,-33.499
C06026=1019.447,267.265,-148.937,-25.604,21.284,-33.269
C06027=1019.437,267.511,-148.985,-25.641,21.295,-33.037
C06028=1019.429,267.756,-149.034,-25.677,21.306,-32.805
C06029=1019.420,268.001,-149.083,-25.714,21.319,-32.571
C06030=1019.409,268.280,-149.140,-25.755,21.333,-32.307
C06031=1019.397,268.559,-149.197,-25.797,21.350,-32.039
C06032=1019.385,268.837,-149.255,-25.839,21.367,-31.772
C06033=1019.372,269.115,-149.313,-25.881,21.386,-31.502
C06034=1019.360,269.360,-149.365,-25.918,21.402,-31.266
C06035=1019.348,269.604,-149.418,-25.955,21.420,-31.029
C06036=1019.337,269.849,-149.472,-25.992,21.439,-30.791
C06037=1019.324,270.092,-149.525,-26.030,21.459,-30.551
C06038=1019.309,270.371,-149.586,-26.072,21.483,-30.277
C06039=1019.294,270.649,-149.649,-26.115,21.507,-30.003
C06040=1019.278,270.927,-149.713,-26.158,21.533,-29.728
C06041=1019.263,271.205,-149.776,-26.201,21.560,-29.450
C06042=1019.248,271.449,-149.833,-26.238,21.585,-29.208
C06043=1019.233,271.692,-149.890,-26.276,21.610,-28.964
C06044=1019.218,271.935,-149.947,-26.314,21.637,-28.720
C06045=1019.202,272.177,-150.005,-26.351,21.664,-28.476
C06046=1019.184,272.456,-150.071,-26.395,21.697,-28.194
C06047=1019.164,272.734,-150.140,-26.438,21.731,-27.910
C06048=1019.145,273.012,-150.208,-26.481,21.766,-27.626
C06049=1019.125,273.289,-150.277,-26.525,21.803,-27.342
C06050=1019.108,273.531,-150.338,-26.562,21.835,-27.092
C06051=1019.089,273.773,-150.399,-26.600,21.869,-26.841
C06052=1019.071,274.015,-150.461,-26.638,21.904,-26.589
C06053=1019.052,274.257,-150.523,-26.676,21.940,-26.336
C06054=1019.030,274.534,-150.596,-26.720,21.983,-26.043
C06055=1019.007,274.812,-150.669,-26.763,22.027,-25.750
C06056=1018.984,275.090,-150.743,-26.807,22.073,-25.453
C06057=1018.960,275.367,-150.817,-26.851,22.119,-25.156
C06058=1018.940,275.607,-150.883,-26.889,22.162,-24.896
C06059=1018.918,275.848,-150.948,-26.927,22.204,-24.635
C06060=1018.896,276.088,-151.014,-26.965,22.250,-24.373
C06061=1018.875,276.328,-151.082,-27.003,22.295,-24.109
C06062=1018.848,276.605,-151.159,-27.046,22.349,-23.804
C06063=1018.822,276.882,-151.238,-27.090,22.404,-23.496
C06064=1018.795,277.160,-151.317,-27.134,22.462,-23.186
C06065=1018.766,277.437,-151.397,-27.177,22.521,-22.877
C06066=1018.743,277.675,-151.467,-27.215,22.573,-22.606
C06067=1018.718,277.914,-151.538,-27.252,22.626,-22.334
C06068=1018.693,278.153,-151.608,-27.290,22.681,-22.062
C06069=1018.668,278.392,-151.679,-27.327,22.737,-21.789
C06070=1018.637,278.669,-151.763,-27.370,22.804,-21.469
C06071=1018.607,278.945,-151.848,-27.413,22.873,-21.147
C06072=1018.576,279.221,-151.934,-27.456,22.942,-20.824
C06073=1018.545,279.498,-152.019,-27.498,23.014,-20.499
C06074=1018.517,279.734,-152.093,-27.534,23.078,-20.218
C06075=1018.489,279.972,-152.168,-27.570,23.142,-19.936
C06076=1018.460,280.209,-152.243,-27.606,23.208,-19.653
C06077=1018.432,280.445,-152.320,-27.642,23.276,-19.367
C06078=1018.398,280.721,-152.409,-27.684,23.357,-19.031
C06079=1018.363,280.998,-152.499,-27.725,23.440,-18.691
C06080=1018.328,281.273,-152.590,-27.766,23.526,-18.349
C06081=1018.291,281.549,-152.681,-27.807,23.613,-18.004
C06082=1018.261,281.784,-152.761,-27.842,23.690,-17.706
C06083=1018.230,282.019,-152.841,-27.877,23.768,-17.406
C06084=1018.198,282.253,-152.920,-27.911,23.848,-17.104
C06085=1018.166,282.489,-153.001,-27.945,23.929,-16.801
C06086=1018.127,282.764,-153.096,-27.984,24.027,-16.441
C06087=1018.088,283.039,-153.192,-28.023,24.128,-16.079
C06088=1018.048,283.314,-153.290,-28.062,24.232,-15.713
C06089=1018.008,283.588,-153.388,-28.100,24.338,-15.343
C06090=1017.974,283.821,-153.472,-28.132,24.429,-15.026
C06091=1017.939,284.054,-153.556,-28.164,24.524,-14.708
C06092=1017.904,284.286,-153.641,-28.195,24.619,-14.388
C06093=1017.868,284.519,-153.727,-28.226,24.716,-14.065
C06094=1017.824,284.793,-153.828,-28.261,24.835,-13.680
C06095=1017.781,285.067,-153.932,-28.296,24.956,-13.292
C06096=1017.737,285.341,-154.034,-28.330,25.079,-12.901
C06097=1017.692,285.614,-154.139,-28.364,25.204,-12.507
C06098=1017.654,285.845,-154.228,-28.391,25.314,-12.171
C06099=1017.616,286.075,-154.318,-28.418,25.425,-11.832
C06100=1017.577,286.305,-154.407,-28.444,25.537,-11.492
C06101=1017.537,286.535,-154.499,-28.470,25.652,-11.148
C06102=1017.490,286.808,-154.607,-28.499,25.792,-10.737
C06103=1017.441,287.080,-154.716,-28.527,25.936,-10.320
C06104=1017.393,287.353,-154.826,-28.555,26.082,-9.899
C06105=1017.343,287.625,-154.938,-28.581,26.233,-9.471
C06106=1017.301,287.852,-155.031,-28.602,26.363,-9.109
C06107=1017.258,288.080,-155.126,-28.622,26.495,-8.743
C06108=1017.216,288.307,-155.221,-28.641,26.630,-8.372
C06109=1017.172,288.535,-155.316,-28.659,26.767,-7.999
C06110=1017.120,288.806,-155.432,-28.679,26.937,-7.545
C06111=1017.067,289.077,-155.549,-28.698,27.109,-7.088
C06112=1017.013,289.347,-155.666,-28.715,27.285,-6.624
C06113=1016.958,289.617,-155.785,-28.730,27.467,-6.153
C06114=1016.912,289.842,-155.883,-28.742,27.622,-5.757
C06115=1016.866,290.067,-155.984,-28.752,27.779,-5.357
C06116=1016.819,290.291,-156.084,-28.760,27.939,-4.952
C06117=1016.771,290.515,-156.186,-28.767,28.103,-4.544
C06118=1016.714,290.784,-156.308,-28.773,28.305,-4.046
C06119=1016.655,291.053,-156.432,-28.777,28.512,-3.541
C06120=1016.596,291.321,-156.557,-28.778,28.722,-3.030
C06121=1016.535,291.589,-156.683,-28.777,28.937,-2.514
C06122=1016.486,291.811,-156.788,-28.773,29.120,-2.080
C06123=1016.435,292.032,-156.894,-28.768,29.306,-1.642
C06124=1016.384,292.252,-157.000,-28.761,29.494,-1.200
C06125=1016.332,292.473,-157.106,-28.751,29.688,-0.751
C06126=1016.269,292.739,-157.238,-28.736,29.926,-0.203
C06127=1016.204,293.006,-157.369,-28.717,30.168,0.353
C06128=1016.139,293.271,-157.502,-28.695,30.417,0.916
C06129=1016.074,293.537,-157.636,-28.669,30.673,1.490
C06130=1016.019,293.754,-157.747,-28.645,30.886,1.967
C06131=1015.964,293.971,-157.858,-28.617,31.104,2.450
C06132=1015.909,294.188,-157.970,-28.586,31.327,2.940
C06133=1015.853,294.404,-158.083,-28.552,31.552,3.436
C06134=1015.783,294.668,-158.223,-28.506,31.835,4.050
C06135=1015.713,294.932,-158.362,-28.455,32.122,4.672
C06136=1015.643,295.194,-158.504,-28.398,32.417,5.306
C06137=1015.570,295.456,-158.646,-28.335,32.716,5.947
C06138=1015.511,295.668,-158.763,-28.280,32.966,6.479
C06139=1015.452,295.881,-158.880,-28.220,33.220,7.016
C06140=1015.391,296.093,-158.998,-28.156,33.478,7.560
C06141=1015.331,296.306,-159.118,-28.087,33.740,8.111
C06142=1015.255,296.566,-159.266,-27.996,34.068,8.799
C06143=1015.178,296.825,-159.414,-27.897,34.404,9.500
C06144=1015.101,297.084,-159.565,-27.790,34.746,10.213
C06145=1015.023,297.343,-159.716,-27.675,35.094,10.935
C06146=1014.959,297.551,-159.839,-27.576,35.380,11.529
C06147=1014.894,297.758,-159.963,-27.470,35.670,12.129
C06148=1014.829,297.965,-160.088,-27.359,35.964,12.737
C06149=1014.763,298.172,-160.213,-27.241,36.263,13.354
C06150=1014.681,298.429,-160.371,-27.085,36.640,14.133
C06151=1014.598,298.684,-160.529,-26.918,37.024,14.926
C06152=1014.513,298.939,-160.688,-26.741,37.414,15.733
C06153=1014.428,299.193,-160.850,-26.551,37.810,16.553
C06154=1014.359,299.395,-160.979,-26.391,38.132,17.220
C06155=1014.290,299.597,-161.109,-26.221,38.458,17.898
C06156=1014.220,299.799,-161.240,-26.044,38.788,18.586
C06157=1014.149,300.000,-161.373,-25.857,39.121,19.283
///RCONF 0,0,0,0,0,0,0,0,0,0,0,0,0,0,0,0,0,0,0,0,0,0,0,0
C06158=1014.059,300.251,-161.539,-25.611,39.544,20.170
C06159=1013.969,300.502,-161.707,-25.349,39.974,21.077
C06160=1013.877,300.752,-161.876,-25.071,40.409,21.999
C06161=1013.785,301.001,-162.048,-24.778,40.847,22.938
C06162=1013.711,301.197,-162.183,-24.533,41.199,23.695
C06163=1013.637,301.393,-162.320,-24.278,41.553,24.463
C06164=1013.561,301.588,-162.458,-24.010,41.911,25.245
C06165=1013.486,301.782,-162.596,-23.731,42.271,26.037
C06166=1013.389,302.029,-162.773,-23.359,42.732,27.060
C06167=1013.291,302.273,-162.952,-22.967,43.196,28.105
C06168=1013.192,302.517,-163.131,-22.552,43.665,29.173
C06169=1013.092,302.761,-163.312,-22.115,44.137,30.264
C06170=1013.013,302.950,-163.455,-21.757,44.508,31.133
C06171=1012.934,303.138,-163.599,-21.384,44.880,32.017
C06172=1012.853,303.327,-163.743,-20.996,45.254,32.916
C06173=1012.772,303.515,-163.888,-20.592,45.628,33.828
C06174=1012.667,303.755,-164.075,-20.052,46.107,35.019
C06175=1012.562,303.993,-164.264,-19.485,46.587,36.235
C06176=1012.455,304.230,-164.454,-18.890,47.066,37.479
C06177=1012.348,304.467,-164.645,-18.265,47.545,38.750
C06178=1012.263,304.648,-164.794,-17.761,47.914,39.754
C06179=1012.178,304.831,-164.944,-17.237,48.283,40.777
C06180=1012.093,305.012,-165.095,-16.695,48.650,41.816
C06181=1012.007,305.191,-165.246,-16.132,49.015,42.875
C06182=1011.894,305.423,-165.443,-15.372,49.485,44.275
C06183=1011.781,305.655,-165.642,-14.578,49.950,45.708
C06184=1011.666,305.885,-165.843,-13.751,50.408,47.169
C06185=1011.551,306.113,-166.044,-12.888,50.859,48.662
C06186=1011.461,306.287,-166.200,-12.202,51.199,49.829
C06187=1011.372,306.461,-166.356,-11.496,51.534,51.012
C06188=1011.281,306.634,-166.513,-10.767,51.863,52.216
C06189=1011.190,306.806,-166.671,-10.018,52.186,53.439
C06190=1011.070,307.030,-166.879,-9.002,52.599,55.068
C06191=1010.948,307.253,-167.087,-7.948,53.000,56.733
C06192=1010.826,307.475,-167.298,-6.854,53.388,58.434
C06193=1010.703,307.694,-167.509,-5.724,53.761,60.165
C06194=1010.608,307.861,-167.670,-4.837,54.035,61.506
C06195=1010.513,308.025,-167.833,-3.930,54.299,62.863
C06196=1010.418,308.190,-167.997,-2.999,54.554,64.242
C06197=1010.322,308.354,-168.160,-2.047,54.798,65.640
C06198=1010.194,308.569,-168.377,-0.758,55.103,67.512
C06199=1010.065,308.783,-168.596,0.564,55.388,69.411
C06200=1009.935,308.995,-168.816,1.921,55.651,71.337
C06201=1009.804,309.205,-169.037,3.305,55.891,73.285
C06202=1009.705,309.362,-169.204,4.368,56.058,74.769
C06203=1009.604,309.519,-169.371,5.445,56.210,76.262
C06204=1009.497,309.675,-169.536,6.540,56.349,77.770
C06205=1009.385,309.828,-169.696,7.643,56.472,79.281
C06206=1009.237,310.014,-169.890,9.013,56.605,81.145
C06207=1009.081,310.197,-170.076,10.390,56.714,83.009
C06208=1008.917,310.376,-170.258,11.770,56.801,84.865
C06209=1008.746,310.553,-170.432,13.151,56.865,86.713
///RCONF 0,0,0,0,1,0,0,0,0,0,0,0,0,0,0,0,0,0,0,0,0,0,0,0
C06210=1019.364,171.442,-138.011,-24.396,21.392,-41.254
C06211=1019.366,170.972,-137.962,-24.395,21.392,-41.256
C06212=1019.367,170.571,-137.919,-24.395,21.392,-41.260
C06213=1019.368,170.171,-137.877,-24.395,21.392,-41.262
C06214=1019.370,169.770,-137.834,-24.394,21.392,-41.265
C06215=1019.371,169.369,-137.791,-24.394,21.393,-41.267
C06216=1019.372,168.969,-137.749,-24.393,21.393,-41.271
C06217=1019.373,168.568,-137.707,-24.393,21.393,-41.273
C06218=1019.374,168.168,-137.665,-24.393,21.394,-41.275
C06219=1019.376,167.768,-137.622,-24.392,21.394,-41.278
C06220=1019.377,167.367,-137.580,-24.392,21.394,-41.280
C06221=1019.378,166.967,-137.537,-24.391,21.393,-41.284
C06222=1019.380,166.567,-137.496,-24.391,21.395,-41.286
C06223=1019.381,166.166,-137.453,-24.391,21.394,-41.289
C06224=1019.382,165.765,-137.411,-24.390,21.394,-41.291
C06225=1019.384,165.365,-137.369,-24.390,21.395,-41.295
C06226=1019.384,164.965,-137.326,-24.390,21.395,-41.297
C06227=1019.385,164.564,-137.285,-24.389,21.395,-41.300
C06228=1019.386,164.179,-137.244,-24.389,21.395,-41.302
C06229=1019.388,163.989,-137.223,-24.389,21.395,-41.304
C06230=1019.388,163.577,-137.181,-24.388,21.396,-41.306
C06231=1019.390,163.342,-137.156,-24.388,21.395,-41.308
C06232=1019.391,163.088,-137.129,-24.388,21.396,-41.309
C06233=1019.392,162.824,-137.102,-24.388,21.396,-41.311
C06234=1019.392,162.556,-137.073,-24.387,21.396,-41.313
C06235=1019.393,162.285,-137.045,-24.387,21.396,-41.315
C06236=1019.394,162.015,-137.016,-24.387,21.397,-41.317
C06237=1019.395,161.752,-136.989,-24.387,21.397,-41.319
C06238=1019.395,161.501,-136.963,-24.386,21.396,-41.320
C06239=1019.396,161.264,-136.937,-24.386,21.396,-41.322
C06240=1019.397,161.040,-136.914,-24.386,21.397,-41.324
C06241=1019.398,160.827,-136.892,-24.386,21.397,-41.325
C06242=1019.400,160.421,-136.849,-24.385,21.397,-41.328
C06243=1019.401,160.024,-136.807,-24.385,21.397,-41.330
C06244=1019.402,159.624,-136.766,-24.384,21.398,-41.333
C06245=1019.407,159.223,-136.725,-24.384,21.398,-41.335
C06246=1019.413,158.822,-136.687,-24.384,21.397,-41.339
C06247=1019.419,158.420,-136.647,-24.383,21.399,-41.341
C06248=1019.425,158.018,-136.608,-24.383,21.398,-41.344
C06249=1020.027,-124.061,-112.558,-23.938,21.716,-44.627
C06250=1020.022,-124.386,-112.536,-23.938,21.716,-44.630
C06251=1020.016,-124.778,-112.508,-23.937,21.717,-44.636
C06252=1020.011,-125.170,-112.481,-23.936,21.718,-44.642
C06253=1020.005,-125.562,-112.455,-23.936,21.719,-44.647
C06254=1019.999,-125.954,-112.427,-23.935,21.719,-44.652
C06255=1019.994,-126.346,-112.399,-23.934,21.719,-44.658
C06256=1019.988,-126.737,-112.373,-23.934,21.720,-44.664
C06257=1019.983,-127.129,-112.346,-23.933,21.721,-44.669
C06258=1019.976,-127.522,-112.319,-23.932,21.722,-44.675
C06259=1019.971,-127.913,-112.292,-23.932,21.723,-44.680
C06260=1019.965,-128.304,-112.265,-23.931,21.723,-44.686
C06261=1019.958,-128.697,-112.238,-23.930,21.723,-44.691
C06262=1019.953,-129.089,-112.211,-23.929,21.724,-44.697
C06263=1019.947,-129.480,-112.185,-23.929,21.725,-44.703
C06264=1019.941,-129.871,-112.157,-23.928,21.726,-44.708
C06265=1019.934,-130.264,-112.131,-23.927,21.727,-44.714
C06266=1019.929,-130.656,-112.104,-23.926,21.727,-44.719
C06267=1019.923,-131.047,-112.077,-23.926,21.728,-44.725
C06268=1019.916,-131.439,-112.050,-23.925,21.728,-44.730
C06269=1019.911,-131.831,-112.023,-23.924,21.729,-44.736
C06270=1019.905,-132.222,-111.997,-23.924,21.730,-44.741
C06271=1019.898,-132.615,-111.970,-23.923,21.730,-44.747
C06272=1019.892,-133.006,-111.943,-23.922,21.731,-44.752
C06273=1019.886,-133.397,-111.916,-23.922,21.732,-44.758
C06274=1019.879,-133.790,-111.890,-23.921,21.732,-44.763
C06275=1020.092,-139.048,-111.292,-23.921,21.732,-44.763
///USER 0
///POSTYPE ROBOT
///RECTAN
///RCONF 0,0,0,1,1,0,0,0,0,0,0,0,0,0,0,0,0,0,0,0,0,0,0,0
C06276=724.889,-216.680,394.500,-180.000,-0.000,-0.000
//INST
///DATE 2021/06/17 16:00
///ATTR SC,RW,RJ
////FRAME ROBOT
///GROUP1 RB1
NOP
MOVL C00000 V=800.0 PL=0
MOVL C00001 V=800.0 PL=0
MOVL C00002 V=800.0 PL=0
MOVL C00003 V=800.0 PL=0
MOVL C00004 V=800.0 PL=0
MOVL C00005 V=800.0 PL=0
MOVL C00006 V=800.0 PL=0
MOVL C00007 V=800.0 PL=0
MOVL C00008 V=800.0 PL=0
MOVL C00009 V=800.0 PL=0
MOVL C00010 V=800.0 PL=0
MOVL C00011 V=800.0 PL=0
MOVL C00012 V=800.0 PL=0
MOVL C00013 V=800.0 PL=0
MOVL C00014 V=800.0 PL=0
MOVL C00015 V=800.0 PL=0
MOVL C00016 V=800.0 PL=0
MOVL C00017 V=800.0 PL=0
MOVL C00018 V=800.0 PL=0
MOVL C00019 V=800.0 PL=0
MOVL C00020 V=800.0 PL=0
MOVL C00021 V=800.0 PL=0
MOVL C00022 V=800.0 PL=0
MOVL C00023 V=800.0 PL=0
MOVL C00024 V=800.0 PL=0
MOVL C00025 V=800.0 PL=0
MOVL C00026 V=800.0 PL=0
MOVL C00027 V=800.0 PL=0
MOVL C00028 V=800.0 PL=0
MOVL C00029 V=800.0 PL=0
MOVL C00030 V=800.0 PL=0
MOVL C00031 V=800.0 PL=0
MOVL C00032 V=800.0 PL=0
MOVL C00033 V=800.0 PL=0
MOVL C00034 V=800.0 PL=0
MOVL C00035 V=800.0 PL=0
MOVL C00036 V=800.0 PL=0
MOVL C00037 V=800.0 PL=0
MOVL C00038 V=800.0 PL=0
MOVL C00039 V=800.0 PL=0
MOVL C00040 V=800.0 PL=0
MOVL C00041 V=800.0 PL=0
MOVL C00042 V=800.0 PL=0
MOVL C00043 V=800.0 PL=0
MOVL C00044 V=800.0 PL=0
MOVL C00045 V=800.0 PL=0
MOVL C00046 V=800.0 PL=0
MOVL C00047 V=800.0 PL=0
MOVL C00048 V=800.0 PL=0
MOVL C00049 V=800.0 PL=0
MOVL C00050 V=800.0 PL=0
MOVL C00051 V=800.0 PL=0
MOVL C00052 V=800.0 PL=0
MOVL C00053 V=800.0 PL=0
MOVL C00054 V=800.0 PL=0
MOVL C00055 V=800.0 PL=0
MOVL C00056 V=800.0 PL=0
MOVL C00057 V=800.0 PL=0
MOVL C00058 V=800.0 PL=0
MOVL C00059 V=800.0 PL=0
MOVL C00060 V=800.0 PL=0
MOVL C00061 V=800.0 PL=0
MOVL C00062 V=800.0 PL=0
MOVL C00063 V=800.0 PL=0
MOVL C00064 V=800.0 PL=0
MOVL C00065 V=800.0 PL=0
MOVL C00066 V=800.0 PL=0
MOVL C00067 V=800.0 PL=0
MOVL C00068 V=800.0 PL=0
MOVL C00069 V=800.0 PL=0
MOVL C00070 V=800.0 PL=0
MOVL C00071 V=800.0 PL=0
MOVL C00072 V=800.0 PL=0
MOVL C00073 V=800.0 PL=0
MOVL C00074 V=800.0 PL=0
MOVL C00075 V=800.0 PL=0
MOVL C00076 V=800.0 PL=0
MOVL C00077 V=800.0 PL=0
MOVL C00078 V=800.0 PL=0
MOVL C00079 V=800.0 PL=0
MOVL C00080 V=800.0 PL=0
MOVL C00081 V=800.0 PL=0
MOVL C00082 V=800.0 PL=0
MOVL C00083 V=800.0 PL=0
MOVL C00084 V=800.0 PL=0
MOVL C00085 V=800.0 PL=0
MOVL C00086 V=800.0 PL=0
MOVL C00087 V=800.0 PL=0
MOVL C00088 V=800.0 PL=0
MOVL C00089 V=800.0 PL=0
MOVL C00090 V=800.0 PL=0
MOVL C00091 V=800.0 PL=0
MOVL C00092 V=800.0 PL=0
MOVL C00093 V=800.0 PL=0
MOVL C00094 V=800.0 PL=0
MOVL C00095 V=800.0 PL=0
MOVL C00096 V=800.0 PL=0
MOVL C00097 V=800.0 PL=0
MOVL C00098 V=800.0 PL=0
MOVL C00099 V=800.0 PL=0
MOVL C00100 V=800.0 PL=0
MOVL C00101 V=800.0 PL=0
MOVL C00102 V=800.0 PL=0
MOVL C00103 V=800.0 PL=0
MOVL C00104 V=800.0 PL=0
MOVL C00105 V=800.0 PL=0
MOVL C00106 V=800.0 PL=0
MOVL C00107 V=800.0 PL=0
MOVL C00108 V=800.0 PL=0
MOVL C00109 V=800.0 PL=0
MOVL C00110 V=800.0 PL=0
MOVL C00111 V=800.0 PL=0
MOVL C00112 V=800.0 PL=0
MOVL C00113 V=800.0 PL=0
MOVL C00114 V=800.0 PL=0
MOVL C00115 V=800.0 PL=0
MOVL C00116 V=800.0 PL=0
MOVL C00117 V=800.0 PL=0
MOVL C00118 V=800.0 PL=0
MOVL C00119 V=800.0 PL=0
MOVL C00120 V=800.0 PL=0
MOVL C00121 V=800.0 PL=0
MOVL C00122 V=800.0 PL=0
MOVL C00123 V=800.0 PL=0
MOVL C00124 V=800.0 PL=0
MOVL C00125 V=800.0 PL=0
MOVL C00126 V=800.0 PL=0
MOVL C00127 V=800.0 PL=0
MOVL C00128 V=800.0 PL=0
MOVL C00129 V=800.0 PL=0
MOVL C00130 V=800.0 PL=0
MOVL C00131 V=800.0 PL=0
MOVL C00132 V=800.0 PL=0
MOVL C00133 V=800.0 PL=0
MOVL C00134 V=800.0 PL=0
MOVL C00135 V=800.0 PL=0
MOVL C00136 V=800.0 PL=0
MOVL C00137 V=800.0 PL=0
MOVL C00138 V=800.0 PL=0
MOVL C00139 V=800.0 PL=0
MOVL C00140 V=800.0 PL=0
MOVL C00141 V=800.0 PL=0
MOVL C00142 V=800.0 PL=0
MOVL C00143 V=800.0 PL=0
MOVL C00144 V=800.0 PL=0
MOVL C00145 V=800.0 PL=0
MOVL C00146 V=800.0 PL=0
MOVL C00147 V=800.0 PL=0
MOVL C00148 V=800.0 PL=0
MOVL C00149 V=800.0 PL=0
MOVL C00150 V=800.0 PL=0
MOVL C00151 V=800.0 PL=0
MOVL C00152 V=800.0 PL=0
MOVL C00153 V=800.0 PL=0
MOVL C00154 V=800.0 PL=0
MOVL C00155 V=800.0 PL=0
MOVL C00156 V=800.0 PL=0
MOVL C00157 V=800.0 PL=0
MOVL C00158 V=800.0 PL=0
MOVL C00159 V=800.0 PL=0
MOVL C00160 V=800.0 PL=0
MOVL C00161 V=800.0 PL=0
MOVL C00162 V=800.0 PL=0
MOVL C00163 V=800.0 PL=0
MOVL C00164 V=800.0 PL=0
MOVL C00165 V=800.0 PL=0
MOVL C00166 V=800.0 PL=0
MOVL C00167 V=800.0 PL=0
MOVL C00168 V=800.0 PL=0
MOVL C00169 V=800.0 PL=0
MOVL C00170 V=800.0 PL=0
MOVL C00171 V=800.0 PL=0
MOVL C00172 V=800.0 PL=0
MOVL C00173 V=800.0 PL=0
MOVL C00174 V=800.0 PL=0
MOVL C00175 V=800.0 PL=0
MOVL C00176 V=800.0 PL=0
MOVL C00177 V=800.0 PL=0
MOVL C00178 V=800.0 PL=0
MOVL C00179 V=800.0 PL=0
MOVL C00180 V=800.0 PL=0
MOVL C00181 V=800.0 PL=0
MOVL C00182 V=800.0 PL=0
MOVL C00183 V=800.0 PL=0
MOVL C00184 V=800.0 PL=0
MOVL C00185 V=800.0 PL=0
MOVL C00186 V=800.0 PL=0
MOVL C00187 V=800.0 PL=0
MOVL C00188 V=800.0 PL=0
MOVL C00189 V=800.0 PL=0
MOVL C00190 V=800.0 PL=0
MOVL C00191 V=800.0 PL=0
MOVL C00192 V=800.0 PL=0
MOVL C00193 V=800.0 PL=0
MOVL C00194 V=800.0 PL=0
MOVL C00195 V=800.0 PL=0
MOVL C00196 V=800.0 PL=0
MOVL C00197 V=800.0 PL=0
MOVL C00198 V=800.0 PL=0
MOVL C00199 V=800.0 PL=0
MOVL C00200 V=800.0 PL=0
MOVL C00201 V=800.0 PL=0
MOVL C00202 V=800.0 PL=0
MOVL C00203 V=800.0 PL=0
MOVL C00204 V=800.0 PL=0
MOVL C00205 V=800.0 PL=0
MOVL C00206 V=800.0 PL=0
MOVL C00207 V=800.0 PL=0
MOVL C00208 V=800.0 PL=0
MOVL C00209 V=800.0 PL=0
MOVL C00210 V=800.0 PL=0
MOVL C00211 V=800.0 PL=0
MOVL C00212 V=800.0 PL=0
MOVL C00213 V=800.0 PL=0
MOVL C00214 V=800.0 PL=0
MOVL C00215 V=800.0 PL=0
MOVL C00216 V=800.0 PL=0
MOVL C00217 V=800.0 PL=0
MOVL C00218 V=800.0 PL=0
MOVL C00219 V=800.0 PL=0
MOVL C00220 V=800.0 PL=0
MOVL C00221 V=800.0 PL=0
MOVL C00222 V=800.0 PL=0
MOVL C00223 V=800.0 PL=0
MOVL C00224 V=800.0 PL=0
MOVL C00225 V=800.0 PL=0
MOVL C00226 V=800.0 PL=0
MOVL C00227 V=800.0 PL=0
MOVL C00228 V=800.0 PL=0
MOVL C00229 V=800.0 PL=0
MOVL C00230 V=800.0 PL=0
MOVL C00231 V=800.0 PL=0
MOVL C00232 V=800.0 PL=0
MOVL C00233 V=800.0 PL=0
MOVL C00234 V=800.0 PL=0
MOVL C00235 V=800.0 PL=0
MOVL C00236 V=800.0 PL=0
MOVL C00237 V=800.0 PL=0
MOVL C00238 V=800.0 PL=0
MOVL C00239 V=800.0 PL=0
MOVL C00240 V=800.0 PL=0
MOVL C00241 V=800.0 PL=0
MOVL C00242 V=800.0 PL=0
MOVL C00243 V=800.0 PL=0
MOVL C00244 V=800.0 PL=0
MOVL C00245 V=800.0 PL=0
MOVL C00246 V=800.0 PL=0
MOVL C00247 V=800.0 PL=0
MOVL C00248 V=800.0 PL=0
MOVL C00249 V=800.0 PL=0
MOVL C00250 V=800.0 PL=0
MOVL C00251 V=800.0 PL=0
MOVL C00252 V=800.0 PL=0
MOVL C00253 V=800.0 PL=0
MOVL C00254 V=800.0 PL=0
MOVL C00255 V=800.0 PL=0
MOVL C00256 V=800.0 PL=0
MOVL C00257 V=800.0 PL=0
MOVL C00258 V=800.0 PL=0
MOVL C00259 V=800.0 PL=0
MOVL C00260 V=800.0 PL=0
MOVL C00261 V=800.0 PL=0
MOVL C00262 V=800.0 PL=0
MOVL C00263 V=800.0 PL=0
MOVL C00264 V=800.0 PL=0
MOVL C00265 V=800.0 PL=0
MOVL C00266 V=800.0 PL=0
MOVL C00267 V=800.0 PL=0
MOVL C00268 V=800.0 PL=0
MOVL C00269 V=800.0 PL=0
MOVL C00270 V=800.0 PL=0
MOVL C00271 V=800.0 PL=0
MOVL C00272 V=800.0 PL=0
MOVL C00273 V=800.0 PL=0
MOVL C00274 V=800.0 PL=0
MOVL C00275 V=800.0 PL=0
MOVL C00276 V=800.0 PL=0
MOVL C00277 V=800.0 PL=0
MOVL C00278 V=800.0 PL=0
MOVL C00279 V=800.0 PL=0
MOVL C00280 V=800.0 PL=0
MOVL C00281 V=800.0 PL=0
MOVL C00282 V=800.0 PL=0
MOVL C00283 V=800.0 PL=0
MOVL C00284 V=800.0 PL=0
MOVL C00285 V=800.0 PL=0
MOVL C00286 V=800.0 PL=0
MOVL C00287 V=800.0 PL=0
MOVL C00288 V=800.0 PL=0
MOVL C00289 V=800.0 PL=0
MOVL C00290 V=800.0 PL=0
MOVL C00291 V=800.0 PL=0
MOVL C00292 V=800.0 PL=0
MOVL C00293 V=800.0 PL=0
MOVL C00294 V=800.0 PL=0
MOVL C00295 V=800.0 PL=0
MOVL C00296 V=800.0 PL=0
MOVL C00297 V=800.0 PL=0
MOVL C00298 V=800.0 PL=0
MOVL C00299 V=800.0 PL=0
MOVL C00300 V=800.0 PL=0
MOVL C00301 V=800.0 PL=0
MOVL C00302 V=800.0 PL=0
MOVL C00303 V=800.0 PL=0
MOVL C00304 V=800.0 PL=0
MOVL C00305 V=800.0 PL=0
MOVL C00306 V=800.0 PL=0
MOVL C00307 V=800.0 PL=0
MOVL C00308 V=800.0 PL=0
MOVL C00309 V=800.0 PL=0
MOVL C00310 V=800.0 PL=0
MOVL C00311 V=800.0 PL=0
MOVL C00312 V=800.0 PL=0
MOVL C00313 V=800.0 PL=0
MOVL C00314 V=800.0 PL=0
MOVL C00315 V=800.0 PL=0
MOVL C00316 V=800.0 PL=0
MOVL C00317 V=800.0 PL=0
MOVL C00318 V=800.0 PL=0
MOVL C00319 V=800.0 PL=0
MOVL C00320 V=800.0 PL=0
MOVL C00321 V=800.0 PL=0
MOVL C00322 V=800.0 PL=0
MOVL C00323 V=800.0 PL=0
MOVL C00324 V=800.0 PL=0
MOVL C00325 V=800.0 PL=0
MOVL C00326 V=800.0 PL=0
MOVL C00327 V=800.0 PL=0
MOVL C00328 V=800.0 PL=0
MOVL C00329 V=800.0 PL=0
MOVL C00330 V=800.0 PL=0
MOVL C00331 V=800.0 PL=0
MOVL C00332 V=800.0 PL=0
MOVL C00333 V=800.0 PL=0
MOVL C00334 V=800.0 PL=0
MOVL C00335 V=800.0 PL=0
MOVL C00336 V=800.0 PL=0
MOVL C00337 V=800.0 PL=0
MOVL C00338 V=800.0 PL=0
MOVL C00339 V=800.0 PL=0
MOVL C00340 V=800.0 PL=0
MOVL C00341 V=800.0 PL=0
MOVL C00342 V=800.0 PL=0
MOVL C00343 V=800.0 PL=0
MOVL C00344 V=800.0 PL=0
MOVL C00345 V=800.0 PL=0
MOVL C00346 V=800.0 PL=0
MOVL C00347 V=800.0 PL=0
MOVL C00348 V=800.0 PL=0
MOVL C00349 V=800.0 PL=0
MOVL C00350 V=800.0 PL=0
MOVL C00351 V=800.0 PL=0
MOVL C00352 V=800.0 PL=0
MOVL C00353 V=800.0 PL=0
MOVL C00354 V=800.0 PL=0
MOVL C00355 V=800.0 PL=0
MOVL C00356 V=800.0 PL=0
MOVL C00357 V=800.0 PL=0
MOVL C00358 V=800.0 PL=0
MOVL C00359 V=800.0 PL=0
MOVL C00360 V=800.0 PL=0
MOVL C00361 V=800.0 PL=0
MOVL C00362 V=800.0 PL=0
MOVL C00363 V=800.0 PL=0
MOVL C00364 V=800.0 PL=0
MOVL C00365 V=800.0 PL=0
MOVL C00366 V=800.0 PL=0
MOVL C00367 V=800.0 PL=0
MOVL C00368 V=800.0 PL=0
MOVL C00369 V=800.0 PL=0
MOVL C00370 V=800.0 PL=0
MOVL C00371 V=800.0 PL=0
MOVL C00372 V=800.0 PL=0
MOVL C00373 V=800.0 PL=0
MOVL C00374 V=800.0 PL=0
MOVL C00375 V=800.0 PL=0
MOVL C00376 V=800.0 PL=0
MOVL C00377 V=800.0 PL=0
MOVL C00378 V=800.0 PL=0
MOVL C00379 V=800.0 PL=0
MOVL C00380 V=800.0 PL=0
MOVL C00381 V=800.0 PL=0
MOVL C00382 V=800.0 PL=0
MOVL C00383 V=800.0 PL=0
MOVL C00384 V=800.0 PL=0
MOVL C00385 V=800.0 PL=0
MOVL C00386 V=800.0 PL=0
MOVL C00387 V=800.0 PL=0
MOVL C00388 V=800.0 PL=0
MOVL C00389 V=800.0 PL=0
MOVL C00390 V=800.0 PL=0
MOVL C00391 V=800.0 PL=0
MOVL C00392 V=800.0 PL=0
MOVL C00393 V=800.0 PL=0
MOVL C00394 V=800.0 PL=0
MOVL C00395 V=800.0 PL=0
MOVL C00396 V=800.0 PL=0
MOVL C00397 V=800.0 PL=0
MOVL C00398 V=800.0 PL=0
MOVL C00399 V=800.0 PL=0
MOVL C00400 V=800.0 PL=0
MOVL C00401 V=800.0 PL=0
MOVL C00402 V=800.0 PL=0
MOVL C00403 V=800.0 PL=0
MOVL C00404 V=800.0 PL=0
MOVL C00405 V=800.0 PL=0
MOVL C00406 V=800.0 PL=0
MOVL C00407 V=800.0 PL=0
MOVL C00408 V=800.0 PL=0
MOVL C00409 V=800.0 PL=0
MOVL C00410 V=800.0 PL=0
MOVL C00411 V=800.0 PL=0
MOVL C00412 V=800.0 PL=0
MOVL C00413 V=800.0 PL=0
MOVL C00414 V=800.0 PL=0
MOVL C00415 V=800.0 PL=0
MOVL C00416 V=800.0 PL=0
MOVL C00417 V=800.0 PL=0
MOVL C00418 V=800.0 PL=0
MOVL C00419 V=800.0 PL=0
MOVL C00420 V=800.0 PL=0
MOVL C00421 V=800.0 PL=0
MOVL C00422 V=800.0 PL=0
MOVL C00423 V=800.0 PL=0
MOVL C00424 V=800.0 PL=0
MOVL C00425 V=800.0 PL=0
MOVL C00426 V=800.0 PL=0
MOVL C00427 V=800.0 PL=0
MOVL C00428 V=800.0 PL=0
MOVL C00429 V=800.0 PL=0
MOVL C00430 V=800.0 PL=0
MOVL C00431 V=800.0 PL=0
MOVL C00432 V=800.0 PL=0
MOVL C00433 V=800.0 PL=0
MOVL C00434 V=800.0 PL=0
MOVL C00435 V=800.0 PL=0
MOVL C00436 V=800.0 PL=0
MOVL C00437 V=800.0 PL=0
MOVL C00438 V=800.0 PL=0
MOVL C00439 V=800.0 PL=0
MOVL C00440 V=800.0 PL=0
MOVL C00441 V=800.0 PL=0
MOVL C00442 V=800.0 PL=0
MOVL C00443 V=800.0 PL=0
MOVL C00444 V=800.0 PL=0
MOVL C00445 V=800.0 PL=0
MOVL C00446 V=800.0 PL=0
MOVL C00447 V=800.0 PL=0
MOVL C00448 V=800.0 PL=0
MOVL C00449 V=800.0 PL=0
MOVL C00450 V=800.0 PL=0
MOVL C00451 V=800.0 PL=0
MOVL C00452 V=800.0 PL=0
MOVL C00453 V=800.0 PL=0
MOVL C00454 V=800.0 PL=0
MOVL C00455 V=800.0 PL=0
MOVL C00456 V=800.0 PL=0
MOVL C00457 V=800.0 PL=0
MOVL C00458 V=800.0 PL=0
MOVL C00459 V=800.0 PL=0
MOVL C00460 V=800.0 PL=0
MOVL C00461 V=800.0 PL=0
MOVL C00462 V=800.0 PL=0
MOVL C00463 V=800.0 PL=0
MOVL C00464 V=800.0 PL=0
MOVL C00465 V=800.0 PL=0
MOVL C00466 V=800.0 PL=0
MOVL C00467 V=800.0 PL=0
MOVL C00468 V=800.0 PL=0
MOVL C00469 V=800.0 PL=0
MOVL C00470 V=800.0 PL=0
MOVL C00471 V=800.0 PL=0
MOVL C00472 V=800.0 PL=0
MOVL C00473 V=800.0 PL=0
MOVL C00474 V=800.0 PL=0
MOVL C00475 V=800.0 PL=0
MOVL C00476 V=800.0 PL=0
MOVL C00477 V=800.0 PL=0
MOVL C00478 V=800.0 PL=0
MOVL C00479 V=800.0 PL=0
MOVL C00480 V=800.0 PL=0
MOVL C00481 V=800.0 PL=0
MOVL C00482 V=800.0 PL=0
MOVL C00483 V=800.0 PL=0
MOVL C00484 V=800.0 PL=0
MOVL C00485 V=800.0 PL=0
MOVL C00486 V=800.0 PL=0
MOVL C00487 V=800.0 PL=0
MOVL C00488 V=800.0 PL=0
MOVL C00489 V=800.0 PL=0
MOVL C00490 V=800.0 PL=0
MOVL C00491 V=800.0 PL=0
MOVL C00492 V=800.0 PL=0
MOVL C00493 V=800.0 PL=0
MOVL C00494 V=800.0 PL=0
MOVL C00495 V=800.0 PL=0
MOVL C00496 V=800.0 PL=0
MOVL C00497 V=800.0 PL=0
MOVL C00498 V=800.0 PL=0
MOVL C00499 V=800.0 PL=0
MOVL C00500 V=800.0 PL=0
MOVL C00501 V=800.0 PL=0
MOVL C00502 V=800.0 PL=0
MOVL C00503 V=800.0 PL=0
MOVL C00504 V=800.0 PL=0
MOVL C00505 V=800.0 PL=0
MOVL C00506 V=800.0 PL=0
MOVL C00507 V=800.0 PL=0
MOVL C00508 V=800.0 PL=0
MOVL C00509 V=800.0 PL=0
MOVL C00510 V=800.0 PL=0
MOVL C00511 V=800.0 PL=0
MOVL C00512 V=800.0 PL=0
MOVL C00513 V=800.0 PL=0
MOVL C00514 V=800.0 PL=0
MOVL C00515 V=800.0 PL=0
MOVL C00516 V=800.0 PL=0
MOVL C00517 V=800.0 PL=0
MOVL C00518 V=800.0 PL=0
MOVL C00519 V=800.0 PL=0
MOVL C00520 V=800.0 PL=0
MOVL C00521 V=800.0 PL=0
MOVL C00522 V=800.0 PL=0
MOVL C00523 V=800.0 PL=0
MOVL C00524 V=800.0 PL=0
MOVL C00525 V=800.0 PL=0
MOVL C00526 V=800.0 PL=0
MOVL C00527 V=800.0 PL=0
MOVL C00528 V=800.0 PL=0
MOVL C00529 V=800.0 PL=0
MOVL C00530 V=800.0 PL=0
MOVL C00531 V=800.0 PL=0
MOVL C00532 V=800.0 PL=0
MOVL C00533 V=800.0 PL=0
MOVL C00534 V=800.0 PL=0
MOVL C00535 V=800.0 PL=0
MOVL C00536 V=800.0 PL=0
MOVL C00537 V=800.0 PL=0
MOVL C00538 V=800.0 PL=0
MOVL C00539 V=800.0 PL=0
MOVL C00540 V=800.0 PL=0
MOVL C00541 V=800.0 PL=0
MOVL C00542 V=800.0 PL=0
MOVL C00543 V=800.0 PL=0
MOVL C00544 V=800.0 PL=0
MOVL C00545 V=800.0 PL=0
MOVL C00546 V=800.0 PL=0
MOVL C00547 V=800.0 PL=0
MOVL C00548 V=800.0 PL=0
MOVL C00549 V=800.0 PL=0
MOVL C00550 V=800.0 PL=0
MOVL C00551 V=800.0 PL=0
MOVL C00552 V=800.0 PL=0
MOVL C00553 V=800.0 PL=0
MOVL C00554 V=800.0 PL=0
MOVL C00555 V=800.0 PL=0
MOVL C00556 V=800.0 PL=0
MOVL C00557 V=800.0 PL=0
MOVL C00558 V=800.0 PL=0
MOVL C00559 V=800.0 PL=0
MOVL C00560 V=800.0 PL=0
MOVL C00561 V=800.0 PL=0
MOVL C00562 V=800.0 PL=0
MOVL C00563 V=800.0 PL=0
MOVL C00564 V=800.0 PL=0
MOVL C00565 V=800.0 PL=0
MOVL C00566 V=800.0 PL=0
MOVL C00567 V=800.0 PL=0
MOVL C00568 V=800.0 PL=0
MOVL C00569 V=800.0 PL=0
MOVL C00570 V=800.0 PL=0
MOVL C00571 V=800.0 PL=0
MOVL C00572 V=800.0 PL=0
MOVL C00573 V=800.0 PL=0
MOVL C00574 V=800.0 PL=0
MOVL C00575 V=800.0 PL=0
MOVL C00576 V=800.0 PL=0
MOVL C00577 V=800.0 PL=0
MOVL C00578 V=800.0 PL=0
MOVL C00579 V=800.0 PL=0
MOVL C00580 V=800.0 PL=0
MOVL C00581 V=800.0 PL=0
MOVL C00582 V=800.0 PL=0
MOVL C00583 V=800.0 PL=0
MOVL C00584 V=800.0 PL=0
MOVL C00585 V=800.0 PL=0
MOVL C00586 V=800.0 PL=0
MOVL C00587 V=800.0 PL=0
MOVL C00588 V=800.0 PL=0
MOVL C00589 V=800.0 PL=0
MOVL C00590 V=800.0 PL=0
MOVL C00591 V=800.0 PL=0
MOVL C00592 V=800.0 PL=0
MOVL C00593 V=800.0 PL=0
MOVL C00594 V=800.0 PL=0
MOVL C00595 V=800.0 PL=0
MOVL C00596 V=800.0 PL=0
MOVL C00597 V=800.0 PL=0
MOVL C00598 V=800.0 PL=0
MOVL C00599 V=800.0 PL=0
MOVL C00600 V=800.0 PL=0
MOVL C00601 V=800.0 PL=0
MOVL C00602 V=800.0 PL=0
MOVL C00603 V=800.0 PL=0
MOVL C00604 V=800.0 PL=0
MOVL C00605 V=800.0 PL=0
MOVL C00606 V=800.0 PL=0
MOVL C00607 V=800.0 PL=0
MOVL C00608 V=800.0 PL=0
MOVL C00609 V=800.0 PL=0
MOVL C00610 V=800.0 PL=0
MOVL C00611 V=800.0 PL=0
MOVL C00612 V=800.0 PL=0
MOVL C00613 V=800.0 PL=0
MOVL C00614 V=800.0 PL=0
MOVL C00615 V=800.0 PL=0
MOVL C00616 V=800.0 PL=0
MOVL C00617 V=800.0 PL=0
MOVL C00618 V=800.0 PL=0
MOVL C00619 V=800.0 PL=0
MOVL C00620 V=800.0 PL=0
MOVL C00621 V=800.0 PL=0
MOVL C00622 V=800.0 PL=0
MOVL C00623 V=800.0 PL=0
MOVL C00624 V=800.0 PL=0
MOVL C00625 V=800.0 PL=0
MOVL C00626 V=800.0 PL=0
MOVL C00627 V=800.0 PL=0
MOVL C00628 V=800.0 PL=0
MOVL C00629 V=800.0 PL=0
MOVL C00630 V=800.0 PL=0
MOVL C00631 V=800.0 PL=0
MOVL C00632 V=800.0 PL=0
MOVL C00633 V=800.0 PL=0
MOVL C00634 V=800.0 PL=0
MOVL C00635 V=800.0 PL=0
MOVL C00636 V=800.0 PL=0
MOVL C00637 V=800.0 PL=0
MOVL C00638 V=800.0 PL=0
MOVL C00639 V=800.0 PL=0
MOVL C00640 V=800.0 PL=0
MOVL C00641 V=800.0 PL=0
MOVL C00642 V=800.0 PL=0
MOVL C00643 V=800.0 PL=0
MOVL C00644 V=800.0 PL=0
MOVL C00645 V=800.0 PL=0
MOVL C00646 V=800.0 PL=0
MOVL C00647 V=800.0 PL=0
MOVL C00648 V=800.0 PL=0
MOVL C00649 V=800.0 PL=0
MOVL C00650 V=800.0 PL=0
MOVL C00651 V=800.0 PL=0
MOVL C00652 V=800.0 PL=0
MOVL C00653 V=800.0 PL=0
MOVL C00654 V=800.0 PL=0
MOVL C00655 V=800.0 PL=0
MOVL C00656 V=800.0 PL=0
MOVL C00657 V=800.0 PL=0
MOVL C00658 V=800.0 PL=0
MOVL C00659 V=800.0 PL=0
MOVL C00660 V=800.0 PL=0
MOVL C00661 V=800.0 PL=0
MOVL C00662 V=800.0 PL=0
MOVL C00663 V=800.0 PL=0
MOVL C00664 V=800.0 PL=0
MOVL C00665 V=800.0 PL=0
MOVL C00666 V=800.0 PL=0
MOVL C00667 V=800.0 PL=0
MOVL C00668 V=800.0 PL=0
MOVL C00669 V=800.0 PL=0
MOVL C00670 V=800.0 PL=0
MOVL C00671 V=800.0 PL=0
MOVL C00672 V=800.0 PL=0
MOVL C00673 V=800.0 PL=0
MOVL C00674 V=800.0 PL=0
MOVL C00675 V=800.0 PL=0
MOVL C00676 V=800.0 PL=0
MOVL C00677 V=800.0 PL=0
MOVL C00678 V=800.0 PL=0
MOVL C00679 V=800.0 PL=0
MOVL C00680 V=800.0 PL=0
MOVL C00681 V=800.0 PL=0
MOVL C00682 V=800.0 PL=0
MOVL C00683 V=800.0 PL=0
MOVL C00684 V=800.0 PL=0
MOVL C00685 V=800.0 PL=0
MOVL C00686 V=800.0 PL=0
MOVL C00687 V=800.0 PL=0
MOVL C00688 V=800.0 PL=0
MOVL C00689 V=800.0 PL=0
MOVL C00690 V=800.0 PL=0
MOVL C00691 V=800.0 PL=0
MOVL C00692 V=800.0 PL=0
MOVL C00693 V=800.0 PL=0
MOVL C00694 V=800.0 PL=0
MOVL C00695 V=800.0 PL=0
MOVL C00696 V=800.0 PL=0
MOVL C00697 V=800.0 PL=0
MOVL C00698 V=800.0 PL=0
MOVL C00699 V=800.0 PL=0
MOVL C00700 V=800.0 PL=0
MOVL C00701 V=800.0 PL=0
MOVL C00702 V=800.0 PL=0
MOVL C00703 V=800.0 PL=0
MOVL C00704 V=800.0 PL=0
MOVL C00705 V=800.0 PL=0
MOVL C00706 V=800.0 PL=0
MOVL C00707 V=800.0 PL=0
MOVL C00708 V=800.0 PL=0
MOVL C00709 V=800.0 PL=0
MOVL C00710 V=800.0 PL=0
MOVL C00711 V=800.0 PL=0
MOVL C00712 V=800.0 PL=0
MOVL C00713 V=800.0 PL=0
MOVL C00714 V=800.0 PL=0
MOVL C00715 V=800.0 PL=0
MOVL C00716 V=800.0 PL=0
MOVL C00717 V=800.0 PL=0
MOVL C00718 V=800.0 PL=0
MOVL C00719 V=800.0 PL=0
MOVL C00720 V=800.0 PL=0
MOVL C00721 V=800.0 PL=0
MOVL C00722 V=800.0 PL=0
MOVL C00723 V=800.0 PL=0
MOVL C00724 V=800.0 PL=0
MOVL C00725 V=800.0 PL=0
MOVL C00726 V=800.0 PL=0
MOVL C00727 V=800.0 PL=0
MOVL C00728 V=800.0 PL=0
MOVL C00729 V=800.0 PL=0
MOVL C00730 V=800.0 PL=0
MOVL C00731 V=800.0 PL=0
MOVL C00732 V=800.0 PL=0
MOVL C00733 V=800.0 PL=0
MOVL C00734 V=800.0 PL=0
MOVL C00735 V=800.0 PL=0
MOVL C00736 V=800.0 PL=0
MOVL C00737 V=800.0 PL=0
MOVL C00738 V=800.0 PL=0
MOVL C00739 V=800.0 PL=0
MOVL C00740 V=800.0 PL=0
MOVL C00741 V=800.0 PL=0
MOVL C00742 V=800.0 PL=0
MOVL C00743 V=800.0 PL=0
MOVL C00744 V=800.0 PL=0
MOVL C00745 V=800.0 PL=0
MOVL C00746 V=800.0 PL=0
MOVL C00747 V=800.0 PL=0
MOVL C00748 V=800.0 PL=0
MOVL C00749 V=800.0 PL=0
MOVL C00750 V=800.0 PL=0
MOVL C00751 V=800.0 PL=0
MOVL C00752 V=800.0 PL=0
MOVL C00753 V=800.0 PL=0
MOVL C00754 V=800.0 PL=0
MOVL C00755 V=800.0 PL=0
MOVL C00756 V=800.0 PL=0
MOVL C00757 V=800.0 PL=0
MOVL C00758 V=800.0 PL=0
MOVL C00759 V=800.0 PL=0
MOVL C00760 V=800.0 PL=0
MOVL C00761 V=800.0 PL=0
MOVL C00762 V=800.0 PL=0
MOVL C00763 V=800.0 PL=0
MOVL C00764 V=800.0 PL=0
MOVL C00765 V=800.0 PL=0
MOVL C00766 V=800.0 PL=0
MOVL C00767 V=800.0 PL=0
MOVL C00768 V=800.0 PL=0
MOVL C00769 V=800.0 PL=0
MOVL C00770 V=800.0 PL=0
MOVL C00771 V=800.0 PL=0
MOVL C00772 V=800.0 PL=0
MOVL C00773 V=800.0 PL=0
MOVL C00774 V=800.0 PL=0
MOVL C00775 V=800.0 PL=0
MOVL C00776 V=800.0 PL=0
MOVL C00777 V=800.0 PL=0
MOVL C00778 V=800.0 PL=0
MOVL C00779 V=800.0 PL=0
MOVL C00780 V=800.0 PL=0
MOVL C00781 V=800.0 PL=0
MOVL C00782 V=800.0 PL=0
MOVL C00783 V=800.0 PL=0
MOVL C00784 V=800.0 PL=0
MOVL C00785 V=800.0 PL=0
MOVL C00786 V=800.0 PL=0
MOVL C00787 V=800.0 PL=0
MOVL C00788 V=800.0 PL=0
MOVL C00789 V=800.0 PL=0
MOVL C00790 V=800.0 PL=0
MOVL C00791 V=800.0 PL=0
MOVL C00792 V=800.0 PL=0
MOVL C00793 V=800.0 PL=0
MOVL C00794 V=800.0 PL=0
MOVL C00795 V=800.0 PL=0
MOVL C00796 V=800.0 PL=0
MOVL C00797 V=800.0 PL=0
MOVL C00798 V=800.0 PL=0
MOVL C00799 V=800.0 PL=0
MOVL C00800 V=800.0 PL=0
MOVL C00801 V=800.0 PL=0
MOVL C00802 V=800.0 PL=0
MOVL C00803 V=800.0 PL=0
MOVL C00804 V=800.0 PL=0
MOVL C00805 V=800.0 PL=0
MOVL C00806 V=800.0 PL=0
MOVL C00807 V=800.0 PL=0
MOVL C00808 V=800.0 PL=0
MOVL C00809 V=800.0 PL=0
MOVL C00810 V=800.0 PL=0
MOVL C00811 V=800.0 PL=0
MOVL C00812 V=800.0 PL=0
MOVL C00813 V=800.0 PL=0
MOVL C00814 V=800.0 PL=0
MOVL C00815 V=800.0 PL=0
MOVL C00816 V=800.0 PL=0
MOVL C00817 V=800.0 PL=0
MOVL C00818 V=800.0 PL=0
MOVL C00819 V=800.0 PL=0
MOVL C00820 V=800.0 PL=0
MOVL C00821 V=800.0 PL=0
MOVL C00822 V=800.0 PL=0
MOVL C00823 V=800.0 PL=0
MOVL C00824 V=800.0 PL=0
MOVL C00825 V=800.0 PL=0
MOVL C00826 V=800.0 PL=0
MOVL C00827 V=800.0 PL=0
MOVL C00828 V=800.0 PL=0
MOVL C00829 V=800.0 PL=0
MOVL C00830 V=800.0 PL=0
MOVL C00831 V=800.0 PL=0
MOVL C00832 V=800.0 PL=0
MOVL C00833 V=800.0 PL=0
MOVL C00834 V=800.0 PL=0
MOVL C00835 V=800.0 PL=0
MOVL C00836 V=800.0 PL=0
MOVL C00837 V=800.0 PL=0
MOVL C00838 V=800.0 PL=0
MOVL C00839 V=800.0 PL=0
MOVL C00840 V=800.0 PL=0
MOVL C00841 V=800.0 PL=0
MOVL C00842 V=800.0 PL=0
MOVL C00843 V=800.0 PL=0
MOVL C00844 V=800.0 PL=0
MOVL C00845 V=800.0 PL=0
MOVL C00846 V=800.0 PL=0
MOVL C00847 V=800.0 PL=0
MOVL C00848 V=800.0 PL=0
MOVL C00849 V=800.0 PL=0
MOVL C00850 V=800.0 PL=0
MOVL C00851 V=800.0 PL=0
MOVL C00852 V=800.0 PL=0
MOVL C00853 V=800.0 PL=0
MOVL C00854 V=800.0 PL=0
MOVL C00855 V=800.0 PL=0
MOVL C00856 V=800.0 PL=0
MOVL C00857 V=800.0 PL=0
MOVL C00858 V=800.0 PL=0
MOVL C00859 V=800.0 PL=0
MOVL C00860 V=800.0 PL=0
MOVL C00861 V=800.0 PL=0
MOVL C00862 V=800.0 PL=0
MOVL C00863 V=800.0 PL=0
MOVL C00864 V=800.0 PL=0
MOVL C00865 V=800.0 PL=0
MOVL C00866 V=800.0 PL=0
MOVL C00867 V=800.0 PL=0
MOVL C00868 V=800.0 PL=0
MOVL C00869 V=800.0 PL=0
MOVL C00870 V=800.0 PL=0
MOVL C00871 V=800.0 PL=0
MOVL C00872 V=800.0 PL=0
MOVL C00873 V=800.0 PL=0
MOVL C00874 V=800.0 PL=0
MOVL C00875 V=800.0 PL=0
MOVL C00876 V=800.0 PL=0
MOVL C00877 V=800.0 PL=0
MOVL C00878 V=800.0 PL=0
MOVL C00879 V=800.0 PL=0
MOVL C00880 V=800.0 PL=0
MOVL C00881 V=800.0 PL=0
MOVL C00882 V=800.0 PL=0
MOVL C00883 V=800.0 PL=0
MOVL C00884 V=800.0 PL=0
MOVL C00885 V=800.0 PL=0
MOVL C00886 V=800.0 PL=0
MOVL C00887 V=800.0 PL=0
MOVL C00888 V=800.0 PL=0
MOVL C00889 V=800.0 PL=0
MOVL C00890 V=800.0 PL=0
MOVL C00891 V=800.0 PL=0
MOVL C00892 V=800.0 PL=0
MOVL C00893 V=800.0 PL=0
MOVL C00894 V=800.0 PL=0
MOVL C00895 V=800.0 PL=0
MOVL C00896 V=800.0 PL=0
MOVL C00897 V=800.0 PL=0
MOVL C00898 V=800.0 PL=0
MOVL C00899 V=800.0 PL=0
MOVL C00900 V=800.0 PL=0
MOVL C00901 V=800.0 PL=0
MOVL C00902 V=800.0 PL=0
MOVL C00903 V=800.0 PL=0
MOVL C00904 V=800.0 PL=0
MOVL C00905 V=800.0 PL=0
MOVL C00906 V=800.0 PL=0
MOVL C00907 V=800.0 PL=0
MOVL C00908 V=800.0 PL=0
MOVL C00909 V=800.0 PL=0
MOVL C00910 V=800.0 PL=0
MOVL C00911 V=800.0 PL=0
MOVL C00912 V=800.0 PL=0
MOVL C00913 V=800.0 PL=0
MOVL C00914 V=800.0 PL=0
MOVL C00915 V=800.0 PL=0
MOVL C00916 V=800.0 PL=0
MOVL C00917 V=800.0 PL=0
MOVL C00918 V=800.0 PL=0
MOVL C00919 V=800.0 PL=0
MOVL C00920 V=800.0 PL=0
MOVL C00921 V=800.0 PL=0
MOVL C00922 V=800.0 PL=0
MOVL C00923 V=800.0 PL=0
MOVL C00924 V=800.0 PL=0
MOVL C00925 V=800.0 PL=0
MOVL C00926 V=800.0 PL=0
MOVL C00927 V=800.0 PL=0
MOVL C00928 V=800.0 PL=0
MOVL C00929 V=800.0 PL=0
MOVL C00930 V=800.0 PL=0
MOVL C00931 V=800.0 PL=0
MOVL C00932 V=800.0 PL=0
MOVL C00933 V=800.0 PL=0
MOVL C00934 V=800.0 PL=0
MOVL C00935 V=800.0 PL=0
MOVL C00936 V=800.0 PL=0
MOVL C00937 V=800.0 PL=0
MOVL C00938 V=800.0 PL=0
MOVL C00939 V=800.0 PL=0
MOVL C00940 V=800.0 PL=0
MOVL C00941 V=800.0 PL=0
MOVL C00942 V=800.0 PL=0
MOVL C00943 V=800.0 PL=0
MOVL C00944 V=800.0 PL=0
MOVL C00945 V=800.0 PL=0
MOVL C00946 V=800.0 PL=0
MOVL C00947 V=800.0 PL=0
MOVL C00948 V=800.0 PL=0
MOVL C00949 V=800.0 PL=0
MOVL C00950 V=800.0 PL=0
MOVL C00951 V=800.0 PL=0
MOVL C00952 V=800.0 PL=0
MOVL C00953 V=800.0 PL=0
MOVL C00954 V=800.0 PL=0
MOVL C00955 V=800.0 PL=0
MOVL C00956 V=800.0 PL=0
MOVL C00957 V=800.0 PL=0
MOVL C00958 V=800.0 PL=0
MOVL C00959 V=800.0 PL=0
MOVL C00960 V=800.0 PL=0
MOVL C00961 V=800.0 PL=0
MOVL C00962 V=800.0 PL=0
MOVL C00963 V=800.0 PL=0
MOVL C00964 V=800.0 PL=0
MOVL C00965 V=800.0 PL=0
MOVL C00966 V=800.0 PL=0
MOVL C00967 V=800.0 PL=0
MOVL C00968 V=800.0 PL=0
MOVL C00969 V=800.0 PL=0
MOVL C00970 V=800.0 PL=0
MOVL C00971 V=800.0 PL=0
MOVL C00972 V=800.0 PL=0
MOVL C00973 V=800.0 PL=0
MOVL C00974 V=800.0 PL=0
MOVL C00975 V=800.0 PL=0
MOVL C00976 V=800.0 PL=0
MOVL C00977 V=800.0 PL=0
MOVL C00978 V=800.0 PL=0
MOVL C00979 V=800.0 PL=0
MOVL C00980 V=800.0 PL=0
MOVL C00981 V=800.0 PL=0
MOVL C00982 V=800.0 PL=0
MOVL C00983 V=800.0 PL=0
MOVL C00984 V=800.0 PL=0
MOVL C00985 V=800.0 PL=0
MOVL C00986 V=800.0 PL=0
MOVL C00987 V=800.0 PL=0
MOVL C00988 V=800.0 PL=0
MOVL C00989 V=800.0 PL=0
MOVL C00990 V=800.0 PL=0
MOVL C00991 V=800.0 PL=0
MOVL C00992 V=800.0 PL=0
MOVL C00993 V=800.0 PL=0
MOVL C00994 V=800.0 PL=0
MOVL C00995 V=800.0 PL=0
MOVL C00996 V=800.0 PL=0
MOVL C00997 V=800.0 PL=0
MOVL C00998 V=800.0 PL=0
MOVL C00999 V=800.0 PL=0
MOVL C01000 V=800.0 PL=0
MOVL C01001 V=800.0 PL=0
MOVL C01002 V=800.0 PL=0
MOVL C01003 V=800.0 PL=0
MOVL C01004 V=800.0 PL=0
MOVL C01005 V=800.0 PL=0
MOVL C01006 V=800.0 PL=0
MOVL C01007 V=800.0 PL=0
MOVL C01008 V=800.0 PL=0
MOVL C01009 V=800.0 PL=0
MOVL C01010 V=800.0 PL=0
MOVL C01011 V=800.0 PL=0
MOVL C01012 V=800.0 PL=0
MOVL C01013 V=800.0 PL=0
MOVL C01014 V=800.0 PL=0
MOVL C01015 V=800.0 PL=0
MOVL C01016 V=800.0 PL=0
MOVL C01017 V=800.0 PL=0
MOVL C01018 V=800.0 PL=0
MOVL C01019 V=800.0 PL=0
MOVL C01020 V=800.0 PL=0
MOVL C01021 V=800.0 PL=0
MOVL C01022 V=800.0 PL=0
MOVL C01023 V=800.0 PL=0
MOVL C01024 V=800.0 PL=0
MOVL C01025 V=800.0 PL=0
MOVL C01026 V=800.0 PL=0
MOVL C01027 V=800.0 PL=0
MOVL C01028 V=800.0 PL=0
MOVL C01029 V=800.0 PL=0
MOVL C01030 V=800.0 PL=0
MOVL C01031 V=800.0 PL=0
MOVL C01032 V=800.0 PL=0
MOVL C01033 V=800.0 PL=0
MOVL C01034 V=800.0 PL=0
MOVL C01035 V=800.0 PL=0
MOVL C01036 V=800.0 PL=0
MOVL C01037 V=800.0 PL=0
MOVL C01038 V=800.0 PL=0
MOVL C01039 V=800.0 PL=0
MOVL C01040 V=800.0 PL=0
MOVL C01041 V=800.0 PL=0
MOVL C01042 V=800.0 PL=0
MOVL C01043 V=800.0 PL=0
MOVL C01044 V=800.0 PL=0
MOVL C01045 V=800.0 PL=0
MOVL C01046 V=800.0 PL=0
MOVL C01047 V=800.0 PL=0
MOVL C01048 V=800.0 PL=0
MOVL C01049 V=800.0 PL=0
MOVL C01050 V=800.0 PL=0
MOVL C01051 V=800.0 PL=0
MOVL C01052 V=800.0 PL=0
MOVL C01053 V=800.0 PL=0
MOVL C01054 V=800.0 PL=0
MOVL C01055 V=800.0 PL=0
MOVL C01056 V=800.0 PL=0
MOVL C01057 V=800.0 PL=0
MOVL C01058 V=800.0 PL=0
MOVL C01059 V=800.0 PL=0
MOVL C01060 V=800.0 PL=0
MOVL C01061 V=800.0 PL=0
MOVL C01062 V=800.0 PL=0
MOVL C01063 V=800.0 PL=0
MOVL C01064 V=800.0 PL=0
MOVL C01065 V=800.0 PL=0
MOVL C01066 V=800.0 PL=0
MOVL C01067 V=800.0 PL=0
MOVL C01068 V=800.0 PL=0
MOVL C01069 V=800.0 PL=0
MOVL C01070 V=800.0 PL=0
MOVL C01071 V=800.0 PL=0
MOVL C01072 V=800.0 PL=0
MOVL C01073 V=800.0 PL=0
MOVL C01074 V=800.0 PL=0
MOVL C01075 V=800.0 PL=0
MOVL C01076 V=800.0 PL=0
MOVL C01077 V=800.0 PL=0
MOVL C01078 V=800.0 PL=0
MOVL C01079 V=800.0 PL=0
MOVL C01080 V=800.0 PL=0
MOVL C01081 V=800.0 PL=0
MOVL C01082 V=800.0 PL=0
MOVL C01083 V=800.0 PL=0
MOVL C01084 V=800.0 PL=0
MOVL C01085 V=800.0 PL=0
MOVL C01086 V=800.0 PL=0
MOVL C01087 V=800.0 PL=0
MOVL C01088 V=800.0 PL=0
MOVL C01089 V=800.0 PL=0
MOVL C01090 V=800.0 PL=0
MOVL C01091 V=800.0 PL=0
MOVL C01092 V=800.0 PL=0
MOVL C01093 V=800.0 PL=0
MOVL C01094 V=800.0 PL=0
MOVL C01095 V=800.0 PL=0
MOVL C01096 V=800.0 PL=0
MOVL C01097 V=800.0 PL=0
MOVL C01098 V=800.0 PL=0
MOVL C01099 V=800.0 PL=0
MOVL C01100 V=800.0 PL=0
MOVL C01101 V=800.0 PL=0
MOVL C01102 V=800.0 PL=0
MOVL C01103 V=800.0 PL=0
MOVL C01104 V=800.0 PL=0
MOVL C01105 V=800.0 PL=0
MOVL C01106 V=800.0 PL=0
MOVL C01107 V=800.0 PL=0
MOVL C01108 V=800.0 PL=0
MOVL C01109 V=800.0 PL=0
MOVL C01110 V=800.0 PL=0
MOVL C01111 V=800.0 PL=0
MOVL C01112 V=800.0 PL=0
MOVL C01113 V=800.0 PL=0
MOVL C01114 V=800.0 PL=0
MOVL C01115 V=800.0 PL=0
MOVL C01116 V=800.0 PL=0
MOVL C01117 V=800.0 PL=0
MOVL C01118 V=800.0 PL=0
MOVL C01119 V=800.0 PL=0
MOVL C01120 V=800.0 PL=0
MOVL C01121 V=800.0 PL=0
MOVL C01122 V=800.0 PL=0
MOVL C01123 V=800.0 PL=0
MOVL C01124 V=800.0 PL=0
MOVL C01125 V=800.0 PL=0
MOVL C01126 V=800.0 PL=0
MOVL C01127 V=800.0 PL=0
MOVL C01128 V=800.0 PL=0
MOVL C01129 V=800.0 PL=0
MOVL C01130 V=800.0 PL=0
MOVL C01131 V=800.0 PL=0
MOVL C01132 V=800.0 PL=0
MOVL C01133 V=800.0 PL=0
MOVL C01134 V=800.0 PL=0
MOVL C01135 V=800.0 PL=0
MOVL C01136 V=800.0 PL=0
MOVL C01137 V=800.0 PL=0
MOVL C01138 V=800.0 PL=0
MOVL C01139 V=800.0 PL=0
MOVL C01140 V=800.0 PL=0
MOVL C01141 V=800.0 PL=0
MOVL C01142 V=800.0 PL=0
MOVL C01143 V=800.0 PL=0
MOVL C01144 V=800.0 PL=0
MOVL C01145 V=800.0 PL=0
MOVL C01146 V=800.0 PL=0
MOVL C01147 V=800.0 PL=0
MOVL C01148 V=800.0 PL=0
MOVL C01149 V=800.0 PL=0
MOVL C01150 V=800.0 PL=0
MOVL C01151 V=800.0 PL=0
MOVL C01152 V=800.0 PL=0
MOVL C01153 V=800.0 PL=0
MOVL C01154 V=800.0 PL=0
MOVL C01155 V=800.0 PL=0
MOVL C01156 V=800.0 PL=0
MOVL C01157 V=800.0 PL=0
MOVL C01158 V=800.0 PL=0
MOVL C01159 V=800.0 PL=0
MOVL C01160 V=800.0 PL=0
MOVL C01161 V=800.0 PL=0
MOVL C01162 V=800.0 PL=0
MOVL C01163 V=800.0 PL=0
MOVL C01164 V=800.0 PL=0
MOVL C01165 V=800.0 PL=0
MOVL C01166 V=800.0 PL=0
MOVL C01167 V=800.0 PL=0
MOVL C01168 V=800.0 PL=0
MOVL C01169 V=800.0 PL=0
MOVL C01170 V=800.0 PL=0
MOVL C01171 V=800.0 PL=0
MOVL C01172 V=800.0 PL=0
MOVL C01173 V=800.0 PL=0
MOVL C01174 V=800.0 PL=0
MOVL C01175 V=800.0 PL=0
MOVL C01176 V=800.0 PL=0
MOVL C01177 V=800.0 PL=0
MOVL C01178 V=800.0 PL=0
MOVL C01179 V=800.0 PL=0
MOVL C01180 V=800.0 PL=0
MOVL C01181 V=800.0 PL=0
MOVL C01182 V=800.0 PL=0
MOVL C01183 V=800.0 PL=0
MOVL C01184 V=800.0 PL=0
MOVL C01185 V=800.0 PL=0
MOVL C01186 V=800.0 PL=0
MOVL C01187 V=800.0 PL=0
MOVL C01188 V=800.0 PL=0
MOVL C01189 V=800.0 PL=0
MOVL C01190 V=800.0 PL=0
MOVL C01191 V=800.0 PL=0
MOVL C01192 V=800.0 PL=0
MOVL C01193 V=800.0 PL=0
MOVL C01194 V=800.0 PL=0
MOVL C01195 V=800.0 PL=0
MOVL C01196 V=800.0 PL=0
MOVL C01197 V=800.0 PL=0
MOVL C01198 V=800.0 PL=0
MOVL C01199 V=800.0 PL=0
MOVL C01200 V=800.0 PL=0
MOVL C01201 V=800.0 PL=0
MOVL C01202 V=800.0 PL=0
MOVL C01203 V=800.0 PL=0
MOVL C01204 V=800.0 PL=0
MOVL C01205 V=800.0 PL=0
MOVL C01206 V=800.0 PL=0
MOVL C01207 V=800.0 PL=0
MOVL C01208 V=800.0 PL=0
MOVL C01209 V=800.0 PL=0
MOVL C01210 V=800.0 PL=0
MOVL C01211 V=800.0 PL=0
MOVL C01212 V=800.0 PL=0
MOVL C01213 V=800.0 PL=0
MOVL C01214 V=800.0 PL=0
MOVL C01215 V=800.0 PL=0
MOVL C01216 V=800.0 PL=0
MOVL C01217 V=800.0 PL=0
MOVL C01218 V=800.0 PL=0
MOVL C01219 V=800.0 PL=0
MOVL C01220 V=800.0 PL=0
MOVL C01221 V=800.0 PL=0
MOVL C01222 V=800.0 PL=0
MOVL C01223 V=800.0 PL=0
MOVL C01224 V=800.0 PL=0
MOVL C01225 V=800.0 PL=0
MOVL C01226 V=800.0 PL=0
MOVL C01227 V=800.0 PL=0
MOVL C01228 V=800.0 PL=0
MOVL C01229 V=800.0 PL=0
MOVL C01230 V=800.0 PL=0
MOVL C01231 V=800.0 PL=0
MOVL C01232 V=800.0 PL=0
MOVL C01233 V=800.0 PL=0
MOVL C01234 V=800.0 PL=0
MOVL C01235 V=800.0 PL=0
MOVL C01236 V=800.0 PL=0
MOVL C01237 V=800.0 PL=0
MOVL C01238 V=800.0 PL=0
MOVL C01239 V=800.0 PL=0
MOVL C01240 V=800.0 PL=0
MOVL C01241 V=800.0 PL=0
MOVL C01242 V=800.0 PL=0
MOVL C01243 V=800.0 PL=0
MOVL C01244 V=800.0 PL=0
MOVL C01245 V=800.0 PL=0
MOVL C01246 V=800.0 PL=0
MOVL C01247 V=800.0 PL=0
MOVL C01248 V=800.0 PL=0
MOVL C01249 V=800.0 PL=0
MOVL C01250 V=800.0 PL=0
MOVL C01251 V=800.0 PL=0
MOVL C01252 V=800.0 PL=0
MOVL C01253 V=800.0 PL=0
MOVL C01254 V=800.0 PL=0
MOVL C01255 V=800.0 PL=0
MOVL C01256 V=800.0 PL=0
MOVL C01257 V=800.0 PL=0
MOVL C01258 V=800.0 PL=0
MOVL C01259 V=800.0 PL=0
MOVL C01260 V=800.0 PL=0
MOVL C01261 V=800.0 PL=0
MOVL C01262 V=800.0 PL=0
MOVL C01263 V=800.0 PL=0
MOVL C01264 V=800.0 PL=0
MOVL C01265 V=800.0 PL=0
MOVL C01266 V=800.0 PL=0
MOVL C01267 V=800.0 PL=0
MOVL C01268 V=800.0 PL=0
MOVL C01269 V=800.0 PL=0
MOVL C01270 V=800.0 PL=0
MOVL C01271 V=800.0 PL=0
MOVL C01272 V=800.0 PL=0
MOVL C01273 V=800.0 PL=0
MOVL C01274 V=800.0 PL=0
MOVL C01275 V=800.0 PL=0
MOVL C01276 V=800.0 PL=0
MOVL C01277 V=800.0 PL=0
MOVL C01278 V=800.0 PL=0
MOVL C01279 V=800.0 PL=0
MOVL C01280 V=800.0 PL=0
MOVL C01281 V=800.0 PL=0
MOVL C01282 V=800.0 PL=0
MOVL C01283 V=800.0 PL=0
MOVL C01284 V=800.0 PL=0
MOVL C01285 V=800.0 PL=0
MOVL C01286 V=800.0 PL=0
MOVL C01287 V=800.0 PL=0
MOVL C01288 V=800.0 PL=0
MOVL C01289 V=800.0 PL=0
MOVL C01290 V=800.0 PL=0
MOVL C01291 V=800.0 PL=0
MOVL C01292 V=800.0 PL=0
MOVL C01293 V=800.0 PL=0
MOVL C01294 V=800.0 PL=0
MOVL C01295 V=800.0 PL=0
MOVL C01296 V=800.0 PL=0
MOVL C01297 V=800.0 PL=0
MOVL C01298 V=800.0 PL=0
MOVL C01299 V=800.0 PL=0
MOVL C01300 V=800.0 PL=0
MOVL C01301 V=800.0 PL=0
MOVL C01302 V=800.0 PL=0
MOVL C01303 V=800.0 PL=0
MOVL C01304 V=800.0 PL=0
MOVL C01305 V=800.0 PL=0
MOVL C01306 V=800.0 PL=0
MOVL C01307 V=800.0 PL=0
MOVL C01308 V=800.0 PL=0
MOVL C01309 V=800.0 PL=0
MOVL C01310 V=800.0 PL=0
MOVL C01311 V=800.0 PL=0
MOVL C01312 V=800.0 PL=0
MOVL C01313 V=800.0 PL=0
MOVL C01314 V=800.0 PL=0
MOVL C01315 V=800.0 PL=0
MOVL C01316 V=800.0 PL=0
MOVL C01317 V=800.0 PL=0
MOVL C01318 V=800.0 PL=0
MOVL C01319 V=800.0 PL=0
MOVL C01320 V=800.0 PL=0
MOVL C01321 V=800.0 PL=0
MOVL C01322 V=800.0 PL=0
MOVL C01323 V=800.0 PL=0
MOVL C01324 V=800.0 PL=0
MOVL C01325 V=800.0 PL=0
MOVL C01326 V=800.0 PL=0
MOVL C01327 V=800.0 PL=0
MOVL C01328 V=800.0 PL=0
MOVL C01329 V=800.0 PL=0
MOVL C01330 V=800.0 PL=0
MOVL C01331 V=800.0 PL=0
MOVL C01332 V=800.0 PL=0
MOVL C01333 V=800.0 PL=0
MOVL C01334 V=800.0 PL=0
MOVL C01335 V=800.0 PL=0
MOVL C01336 V=800.0 PL=0
MOVL C01337 V=800.0 PL=0
MOVL C01338 V=800.0 PL=0
MOVL C01339 V=800.0 PL=0
MOVL C01340 V=800.0 PL=0
MOVL C01341 V=800.0 PL=0
MOVL C01342 V=800.0 PL=0
MOVL C01343 V=800.0 PL=0
MOVL C01344 V=800.0 PL=0
MOVL C01345 V=800.0 PL=0
MOVL C01346 V=800.0 PL=0
MOVL C01347 V=800.0 PL=0
MOVL C01348 V=800.0 PL=0
MOVL C01349 V=800.0 PL=0
MOVL C01350 V=800.0 PL=0
MOVL C01351 V=800.0 PL=0
MOVL C01352 V=800.0 PL=0
MOVL C01353 V=800.0 PL=0
MOVL C01354 V=800.0 PL=0
MOVL C01355 V=800.0 PL=0
MOVL C01356 V=800.0 PL=0
MOVL C01357 V=800.0 PL=0
MOVL C01358 V=800.0 PL=0
MOVL C01359 V=800.0 PL=0
MOVL C01360 V=800.0 PL=0
MOVL C01361 V=800.0 PL=0
MOVL C01362 V=800.0 PL=0
MOVL C01363 V=800.0 PL=0
MOVL C01364 V=800.0 PL=0
MOVL C01365 V=800.0 PL=0
MOVL C01366 V=800.0 PL=0
MOVL C01367 V=800.0 PL=0
MOVL C01368 V=800.0 PL=0
MOVL C01369 V=800.0 PL=0
MOVL C01370 V=800.0 PL=0
MOVL C01371 V=800.0 PL=0
MOVL C01372 V=800.0 PL=0
MOVL C01373 V=800.0 PL=0
MOVL C01374 V=800.0 PL=0
MOVL C01375 V=800.0 PL=0
MOVL C01376 V=800.0 PL=0
MOVL C01377 V=800.0 PL=0
MOVL C01378 V=800.0 PL=0
MOVL C01379 V=800.0 PL=0
MOVL C01380 V=800.0 PL=0
MOVL C01381 V=800.0 PL=0
MOVL C01382 V=800.0 PL=0
MOVL C01383 V=800.0 PL=0
MOVL C01384 V=800.0 PL=0
MOVL C01385 V=800.0 PL=0
MOVL C01386 V=800.0 PL=0
MOVL C01387 V=800.0 PL=0
MOVL C01388 V=800.0 PL=0
MOVL C01389 V=800.0 PL=0
MOVL C01390 V=800.0 PL=0
MOVL C01391 V=800.0 PL=0
MOVL C01392 V=800.0 PL=0
MOVL C01393 V=800.0 PL=0
MOVL C01394 V=800.0 PL=0
MOVL C01395 V=800.0 PL=0
MOVL C01396 V=800.0 PL=0
MOVL C01397 V=800.0 PL=0
MOVL C01398 V=800.0 PL=0
MOVL C01399 V=800.0 PL=0
MOVL C01400 V=800.0 PL=0
MOVL C01401 V=800.0 PL=0
MOVL C01402 V=800.0 PL=0
MOVL C01403 V=800.0 PL=0
MOVL C01404 V=800.0 PL=0
MOVL C01405 V=800.0 PL=0
MOVL C01406 V=800.0 PL=0
MOVL C01407 V=800.0 PL=0
MOVL C01408 V=800.0 PL=0
MOVL C01409 V=800.0 PL=0
MOVL C01410 V=800.0 PL=0
MOVL C01411 V=800.0 PL=0
MOVL C01412 V=800.0 PL=0
MOVL C01413 V=800.0 PL=0
MOVL C01414 V=800.0 PL=0
MOVL C01415 V=800.0 PL=0
MOVL C01416 V=800.0 PL=0
MOVL C01417 V=800.0 PL=0
MOVL C01418 V=800.0 PL=0
MOVL C01419 V=800.0 PL=0
MOVL C01420 V=800.0 PL=0
MOVL C01421 V=800.0 PL=0
MOVL C01422 V=800.0 PL=0
MOVL C01423 V=800.0 PL=0
MOVL C01424 V=800.0 PL=0
MOVL C01425 V=800.0 PL=0
MOVL C01426 V=800.0 PL=0
MOVL C01427 V=800.0 PL=0
MOVL C01428 V=800.0 PL=0
MOVL C01429 V=800.0 PL=0
MOVL C01430 V=800.0 PL=0
MOVL C01431 V=800.0 PL=0
MOVL C01432 V=800.0 PL=0
MOVL C01433 V=800.0 PL=0
MOVL C01434 V=800.0 PL=0
MOVL C01435 V=800.0 PL=0
MOVL C01436 V=800.0 PL=0
MOVL C01437 V=800.0 PL=0
MOVL C01438 V=800.0 PL=0
MOVL C01439 V=800.0 PL=0
MOVL C01440 V=800.0 PL=0
MOVL C01441 V=800.0 PL=0
MOVL C01442 V=800.0 PL=0
MOVL C01443 V=800.0 PL=0
MOVL C01444 V=800.0 PL=0
MOVL C01445 V=800.0 PL=0
MOVL C01446 V=800.0 PL=0
MOVL C01447 V=800.0 PL=0
MOVL C01448 V=800.0 PL=0
MOVL C01449 V=800.0 PL=0
MOVL C01450 V=800.0 PL=0
MOVL C01451 V=800.0 PL=0
MOVL C01452 V=800.0 PL=0
MOVL C01453 V=800.0 PL=0
MOVL C01454 V=800.0 PL=0
MOVL C01455 V=800.0 PL=0
MOVL C01456 V=800.0 PL=0
MOVL C01457 V=800.0 PL=0
MOVL C01458 V=800.0 PL=0
MOVL C01459 V=800.0 PL=0
MOVL C01460 V=800.0 PL=0
MOVL C01461 V=800.0 PL=0
MOVL C01462 V=800.0 PL=0
MOVL C01463 V=800.0 PL=0
MOVL C01464 V=800.0 PL=0
MOVL C01465 V=800.0 PL=0
MOVL C01466 V=800.0 PL=0
MOVL C01467 V=800.0 PL=0
MOVL C01468 V=800.0 PL=0
MOVL C01469 V=800.0 PL=0
MOVL C01470 V=800.0 PL=0
MOVL C01471 V=800.0 PL=0
MOVL C01472 V=800.0 PL=0
MOVL C01473 V=800.0 PL=0
MOVL C01474 V=800.0 PL=0
MOVL C01475 V=800.0 PL=0
MOVL C01476 V=800.0 PL=0
MOVL C01477 V=800.0 PL=0
MOVL C01478 V=800.0 PL=0
MOVL C01479 V=800.0 PL=0
MOVL C01480 V=800.0 PL=0
MOVL C01481 V=800.0 PL=0
MOVL C01482 V=800.0 PL=0
MOVL C01483 V=800.0 PL=0
MOVL C01484 V=800.0 PL=0
MOVL C01485 V=800.0 PL=0
MOVL C01486 V=800.0 PL=0
MOVL C01487 V=800.0 PL=0
MOVL C01488 V=800.0 PL=0
MOVL C01489 V=800.0 PL=0
MOVL C01490 V=800.0 PL=0
MOVL C01491 V=800.0 PL=0
MOVL C01492 V=800.0 PL=0
MOVL C01493 V=800.0 PL=0
MOVL C01494 V=800.0 PL=0
MOVL C01495 V=800.0 PL=0
MOVL C01496 V=800.0 PL=0
MOVL C01497 V=800.0 PL=0
MOVL C01498 V=800.0 PL=0
MOVL C01499 V=800.0 PL=0
MOVL C01500 V=800.0 PL=0
MOVL C01501 V=800.0 PL=0
MOVL C01502 V=800.0 PL=0
MOVL C01503 V=800.0 PL=0
MOVL C01504 V=800.0 PL=0
MOVL C01505 V=800.0 PL=0
MOVL C01506 V=800.0 PL=0
MOVL C01507 V=800.0 PL=0
MOVL C01508 V=800.0 PL=0
MOVL C01509 V=800.0 PL=0
MOVL C01510 V=800.0 PL=0
MOVL C01511 V=800.0 PL=0
MOVL C01512 V=800.0 PL=0
MOVL C01513 V=800.0 PL=0
MOVL C01514 V=800.0 PL=0
MOVL C01515 V=800.0 PL=0
MOVL C01516 V=800.0 PL=0
MOVL C01517 V=800.0 PL=0
MOVL C01518 V=800.0 PL=0
MOVL C01519 V=800.0 PL=0
MOVL C01520 V=800.0 PL=0
MOVL C01521 V=800.0 PL=0
MOVL C01522 V=800.0 PL=0
MOVL C01523 V=800.0 PL=0
MOVL C01524 V=800.0 PL=0
MOVL C01525 V=800.0 PL=0
MOVL C01526 V=800.0 PL=0
MOVL C01527 V=800.0 PL=0
MOVL C01528 V=800.0 PL=0
MOVL C01529 V=800.0 PL=0
MOVL C01530 V=800.0 PL=0
MOVL C01531 V=800.0 PL=0
MOVL C01532 V=800.0 PL=0
MOVL C01533 V=800.0 PL=0
MOVL C01534 V=800.0 PL=0
MOVL C01535 V=800.0 PL=0
MOVL C01536 V=800.0 PL=0
MOVL C01537 V=800.0 PL=0
MOVL C01538 V=800.0 PL=0
MOVL C01539 V=800.0 PL=0
MOVL C01540 V=800.0 PL=0
MOVL C01541 V=800.0 PL=0
MOVL C01542 V=800.0 PL=0
MOVL C01543 V=800.0 PL=0
MOVL C01544 V=800.0 PL=0
MOVL C01545 V=800.0 PL=0
MOVL C01546 V=800.0 PL=0
MOVL C01547 V=800.0 PL=0
MOVL C01548 V=800.0 PL=0
MOVL C01549 V=800.0 PL=0
MOVL C01550 V=800.0 PL=0
MOVL C01551 V=800.0 PL=0
MOVL C01552 V=800.0 PL=0
MOVL C01553 V=800.0 PL=0
MOVL C01554 V=800.0 PL=0
MOVL C01555 V=800.0 PL=0
MOVL C01556 V=800.0 PL=0
MOVL C01557 V=800.0 PL=0
MOVL C01558 V=800.0 PL=0
MOVL C01559 V=800.0 PL=0
MOVL C01560 V=800.0 PL=0
MOVL C01561 V=800.0 PL=0
MOVL C01562 V=800.0 PL=0
MOVL C01563 V=800.0 PL=0
MOVL C01564 V=800.0 PL=0
MOVL C01565 V=800.0 PL=0
MOVL C01566 V=800.0 PL=0
MOVL C01567 V=800.0 PL=0
MOVL C01568 V=800.0 PL=0
MOVL C01569 V=800.0 PL=0
MOVL C01570 V=800.0 PL=0
MOVL C01571 V=800.0 PL=0
MOVL C01572 V=800.0 PL=0
MOVL C01573 V=800.0 PL=0
MOVL C01574 V=800.0 PL=0
MOVL C01575 V=800.0 PL=0
MOVL C01576 V=800.0 PL=0
MOVL C01577 V=800.0 PL=0
MOVL C01578 V=800.0 PL=0
MOVL C01579 V=800.0 PL=0
MOVL C01580 V=800.0 PL=0
MOVL C01581 V=800.0 PL=0
MOVL C01582 V=800.0 PL=0
MOVL C01583 V=800.0 PL=0
MOVL C01584 V=800.0 PL=0
MOVL C01585 V=800.0 PL=0
MOVL C01586 V=800.0 PL=0
MOVL C01587 V=800.0 PL=0
MOVL C01588 V=800.0 PL=0
MOVL C01589 V=800.0 PL=0
MOVL C01590 V=800.0 PL=0
MOVL C01591 V=800.0 PL=0
MOVL C01592 V=800.0 PL=0
MOVL C01593 V=800.0 PL=0
MOVL C01594 V=800.0 PL=0
MOVL C01595 V=800.0 PL=0
MOVL C01596 V=800.0 PL=0
MOVL C01597 V=800.0 PL=0
MOVL C01598 V=800.0 PL=0
MOVL C01599 V=800.0 PL=0
MOVL C01600 V=800.0 PL=0
MOVL C01601 V=800.0 PL=0
MOVL C01602 V=800.0 PL=0
MOVL C01603 V=800.0 PL=0
MOVL C01604 V=800.0 PL=0
MOVL C01605 V=800.0 PL=0
MOVL C01606 V=800.0 PL=0
MOVL C01607 V=800.0 PL=0
MOVL C01608 V=800.0 PL=0
MOVL C01609 V=800.0 PL=0
MOVL C01610 V=800.0 PL=0
MOVL C01611 V=800.0 PL=0
MOVL C01612 V=800.0 PL=0
MOVL C01613 V=800.0 PL=0
MOVL C01614 V=800.0 PL=0
MOVL C01615 V=800.0 PL=0
MOVL C01616 V=800.0 PL=0
MOVL C01617 V=800.0 PL=0
MOVL C01618 V=800.0 PL=0
MOVL C01619 V=800.0 PL=0
MOVL C01620 V=800.0 PL=0
MOVL C01621 V=800.0 PL=0
MOVL C01622 V=800.0 PL=0
MOVL C01623 V=800.0 PL=0
MOVL C01624 V=800.0 PL=0
MOVL C01625 V=800.0 PL=0
MOVL C01626 V=800.0 PL=0
MOVL C01627 V=800.0 PL=0
MOVL C01628 V=800.0 PL=0
MOVL C01629 V=800.0 PL=0
MOVL C01630 V=800.0 PL=0
MOVL C01631 V=800.0 PL=0
MOVL C01632 V=800.0 PL=0
MOVL C01633 V=800.0 PL=0
MOVL C01634 V=800.0 PL=0
MOVL C01635 V=800.0 PL=0
MOVL C01636 V=800.0 PL=0
MOVL C01637 V=800.0 PL=0
MOVL C01638 V=800.0 PL=0
MOVL C01639 V=800.0 PL=0
MOVL C01640 V=800.0 PL=0
MOVL C01641 V=800.0 PL=0
MOVL C01642 V=800.0 PL=0
MOVL C01643 V=800.0 PL=0
MOVL C01644 V=800.0 PL=0
MOVL C01645 V=800.0 PL=0
MOVL C01646 V=800.0 PL=0
MOVL C01647 V=800.0 PL=0
MOVL C01648 V=800.0 PL=0
MOVL C01649 V=800.0 PL=0
MOVL C01650 V=800.0 PL=0
MOVL C01651 V=800.0 PL=0
MOVL C01652 V=800.0 PL=0
MOVL C01653 V=800.0 PL=0
MOVL C01654 V=800.0 PL=0
MOVL C01655 V=800.0 PL=0
MOVL C01656 V=800.0 PL=0
MOVL C01657 V=800.0 PL=0
MOVL C01658 V=800.0 PL=0
MOVL C01659 V=800.0 PL=0
MOVL C01660 V=800.0 PL=0
MOVL C01661 V=800.0 PL=0
MOVL C01662 V=800.0 PL=0
MOVL C01663 V=800.0 PL=0
MOVL C01664 V=800.0 PL=0
MOVL C01665 V=800.0 PL=0
MOVL C01666 V=800.0 PL=0
MOVL C01667 V=800.0 PL=0
MOVL C01668 V=800.0 PL=0
MOVL C01669 V=800.0 PL=0
MOVL C01670 V=800.0 PL=0
MOVL C01671 V=800.0 PL=0
MOVL C01672 V=800.0 PL=0
MOVL C01673 V=800.0 PL=0
MOVL C01674 V=800.0 PL=0
MOVL C01675 V=800.0 PL=0
MOVL C01676 V=800.0 PL=0
MOVL C01677 V=800.0 PL=0
MOVL C01678 V=800.0 PL=0
MOVL C01679 V=800.0 PL=0
MOVL C01680 V=800.0 PL=0
MOVL C01681 V=800.0 PL=0
MOVL C01682 V=800.0 PL=0
MOVL C01683 V=800.0 PL=0
MOVL C01684 V=800.0 PL=0
MOVL C01685 V=800.0 PL=0
MOVL C01686 V=800.0 PL=0
MOVL C01687 V=800.0 PL=0
MOVL C01688 V=800.0 PL=0
MOVL C01689 V=800.0 PL=0
MOVL C01690 V=800.0 PL=0
MOVL C01691 V=800.0 PL=0
MOVL C01692 V=800.0 PL=0
MOVL C01693 V=800.0 PL=0
MOVL C01694 V=800.0 PL=0
MOVL C01695 V=800.0 PL=0
MOVL C01696 V=800.0 PL=0
MOVL C01697 V=800.0 PL=0
MOVL C01698 V=800.0 PL=0
MOVL C01699 V=800.0 PL=0
MOVL C01700 V=800.0 PL=0
MOVL C01701 V=800.0 PL=0
MOVL C01702 V=800.0 PL=0
MOVL C01703 V=800.0 PL=0
MOVL C01704 V=800.0 PL=0
MOVL C01705 V=800.0 PL=0
MOVL C01706 V=800.0 PL=0
MOVL C01707 V=800.0 PL=0
MOVL C01708 V=800.0 PL=0
MOVL C01709 V=800.0 PL=0
MOVL C01710 V=800.0 PL=0
MOVL C01711 V=800.0 PL=0
MOVL C01712 V=800.0 PL=0
MOVL C01713 V=800.0 PL=0
MOVL C01714 V=800.0 PL=0
MOVL C01715 V=800.0 PL=0
MOVL C01716 V=800.0 PL=0
MOVL C01717 V=800.0 PL=0
MOVL C01718 V=800.0 PL=0
MOVL C01719 V=800.0 PL=0
MOVL C01720 V=800.0 PL=0
MOVL C01721 V=800.0 PL=0
MOVL C01722 V=800.0 PL=0
MOVL C01723 V=800.0 PL=0
MOVL C01724 V=800.0 PL=0
MOVL C01725 V=800.0 PL=0
MOVL C01726 V=800.0 PL=0
MOVL C01727 V=800.0 PL=0
MOVL C01728 V=800.0 PL=0
MOVL C01729 V=800.0 PL=0
MOVL C01730 V=800.0 PL=0
MOVL C01731 V=800.0 PL=0
MOVL C01732 V=800.0 PL=0
MOVL C01733 V=800.0 PL=0
MOVL C01734 V=800.0 PL=0
MOVL C01735 V=800.0 PL=0
MOVL C01736 V=800.0 PL=0
MOVL C01737 V=800.0 PL=0
MOVL C01738 V=800.0 PL=0
MOVL C01739 V=800.0 PL=0
MOVL C01740 V=800.0 PL=0
MOVL C01741 V=800.0 PL=0
MOVL C01742 V=800.0 PL=0
MOVL C01743 V=800.0 PL=0
MOVL C01744 V=800.0 PL=0
MOVL C01745 V=800.0 PL=0
MOVL C01746 V=800.0 PL=0
MOVL C01747 V=800.0 PL=0
MOVL C01748 V=800.0 PL=0
MOVL C01749 V=800.0 PL=0
MOVL C01750 V=800.0 PL=0
MOVL C01751 V=800.0 PL=0
MOVL C01752 V=800.0 PL=0
MOVL C01753 V=800.0 PL=0
MOVL C01754 V=800.0 PL=0
MOVL C01755 V=800.0 PL=0
MOVL C01756 V=800.0 PL=0
MOVL C01757 V=800.0 PL=0
MOVL C01758 V=800.0 PL=0
MOVL C01759 V=800.0 PL=0
MOVL C01760 V=800.0 PL=0
MOVL C01761 V=800.0 PL=0
MOVL C01762 V=800.0 PL=0
MOVL C01763 V=800.0 PL=0
MOVL C01764 V=800.0 PL=0
MOVL C01765 V=800.0 PL=0
MOVL C01766 V=800.0 PL=0
MOVL C01767 V=800.0 PL=0
MOVL C01768 V=800.0 PL=0
MOVL C01769 V=800.0 PL=0
MOVL C01770 V=800.0 PL=0
MOVL C01771 V=800.0 PL=0
MOVL C01772 V=800.0 PL=0
MOVL C01773 V=800.0 PL=0
MOVL C01774 V=800.0 PL=0
MOVL C01775 V=800.0 PL=0
MOVL C01776 V=800.0 PL=0
MOVL C01777 V=800.0 PL=0
MOVL C01778 V=800.0 PL=0
MOVL C01779 V=800.0 PL=0
MOVL C01780 V=800.0 PL=0
MOVL C01781 V=800.0 PL=0
MOVL C01782 V=800.0 PL=0
MOVL C01783 V=800.0 PL=0
MOVL C01784 V=800.0 PL=0
MOVL C01785 V=800.0 PL=0
MOVL C01786 V=800.0 PL=0
MOVL C01787 V=800.0 PL=0
MOVL C01788 V=800.0 PL=0
MOVL C01789 V=800.0 PL=0
MOVL C01790 V=800.0 PL=0
MOVL C01791 V=800.0 PL=0
MOVL C01792 V=800.0 PL=0
MOVL C01793 V=800.0 PL=0
MOVL C01794 V=800.0 PL=0
MOVL C01795 V=800.0 PL=0
MOVL C01796 V=800.0 PL=0
MOVL C01797 V=800.0 PL=0
MOVL C01798 V=800.0 PL=0
MOVL C01799 V=800.0 PL=0
MOVL C01800 V=800.0 PL=0
MOVL C01801 V=800.0 PL=0
MOVL C01802 V=800.0 PL=0
MOVL C01803 V=800.0 PL=0
MOVL C01804 V=800.0 PL=0
MOVL C01805 V=800.0 PL=0
MOVL C01806 V=800.0 PL=0
MOVL C01807 V=800.0 PL=0
MOVL C01808 V=800.0 PL=0
MOVL C01809 V=800.0 PL=0
MOVL C01810 V=800.0 PL=0
MOVL C01811 V=800.0 PL=0
MOVL C01812 V=800.0 PL=0
MOVL C01813 V=800.0 PL=0
MOVL C01814 V=800.0 PL=0
MOVL C01815 V=800.0 PL=0
MOVL C01816 V=800.0 PL=0
MOVL C01817 V=800.0 PL=0
MOVL C01818 V=800.0 PL=0
MOVL C01819 V=800.0 PL=0
MOVL C01820 V=800.0 PL=0
MOVL C01821 V=800.0 PL=0
MOVL C01822 V=800.0 PL=0
MOVL C01823 V=800.0 PL=0
MOVL C01824 V=800.0 PL=0
MOVL C01825 V=800.0 PL=0
MOVL C01826 V=800.0 PL=0
MOVL C01827 V=800.0 PL=0
MOVL C01828 V=800.0 PL=0
MOVL C01829 V=800.0 PL=0
MOVL C01830 V=800.0 PL=0
MOVL C01831 V=800.0 PL=0
MOVL C01832 V=800.0 PL=0
MOVL C01833 V=800.0 PL=0
MOVL C01834 V=800.0 PL=0
MOVL C01835 V=800.0 PL=0
MOVL C01836 V=800.0 PL=0
MOVL C01837 V=800.0 PL=0
MOVL C01838 V=800.0 PL=0
MOVL C01839 V=800.0 PL=0
MOVL C01840 V=800.0 PL=0
MOVL C01841 V=800.0 PL=0
MOVL C01842 V=800.0 PL=0
MOVL C01843 V=800.0 PL=0
MOVL C01844 V=800.0 PL=0
MOVL C01845 V=800.0 PL=0
MOVL C01846 V=800.0 PL=0
MOVL C01847 V=800.0 PL=0
MOVL C01848 V=800.0 PL=0
MOVL C01849 V=800.0 PL=0
MOVL C01850 V=800.0 PL=0
MOVL C01851 V=800.0 PL=0
MOVL C01852 V=800.0 PL=0
MOVL C01853 V=800.0 PL=0
MOVL C01854 V=800.0 PL=0
MOVL C01855 V=800.0 PL=0
MOVL C01856 V=800.0 PL=0
MOVL C01857 V=800.0 PL=0
MOVL C01858 V=800.0 PL=0
MOVL C01859 V=800.0 PL=0
MOVL C01860 V=800.0 PL=0
MOVL C01861 V=800.0 PL=0
MOVL C01862 V=800.0 PL=0
MOVL C01863 V=800.0 PL=0
MOVL C01864 V=800.0 PL=0
MOVL C01865 V=800.0 PL=0
MOVL C01866 V=800.0 PL=0
MOVL C01867 V=800.0 PL=0
MOVL C01868 V=800.0 PL=0
MOVL C01869 V=800.0 PL=0
MOVL C01870 V=800.0 PL=0
MOVL C01871 V=800.0 PL=0
MOVL C01872 V=800.0 PL=0
MOVL C01873 V=800.0 PL=0
MOVL C01874 V=800.0 PL=0
MOVL C01875 V=800.0 PL=0
MOVL C01876 V=800.0 PL=0
MOVL C01877 V=800.0 PL=0
MOVL C01878 V=800.0 PL=0
MOVL C01879 V=800.0 PL=0
MOVL C01880 V=800.0 PL=0
MOVL C01881 V=800.0 PL=0
MOVL C01882 V=800.0 PL=0
MOVL C01883 V=800.0 PL=0
MOVL C01884 V=800.0 PL=0
MOVL C01885 V=800.0 PL=0
MOVL C01886 V=800.0 PL=0
MOVL C01887 V=800.0 PL=0
MOVL C01888 V=800.0 PL=0
MOVL C01889 V=800.0 PL=0
MOVL C01890 V=800.0 PL=0
MOVL C01891 V=800.0 PL=0
MOVL C01892 V=800.0 PL=0
MOVL C01893 V=800.0 PL=0
MOVL C01894 V=800.0 PL=0
MOVL C01895 V=800.0 PL=0
MOVL C01896 V=800.0 PL=0
MOVL C01897 V=800.0 PL=0
MOVL C01898 V=800.0 PL=0
MOVL C01899 V=800.0 PL=0
MOVL C01900 V=800.0 PL=0
MOVL C01901 V=800.0 PL=0
MOVL C01902 V=800.0 PL=0
MOVL C01903 V=800.0 PL=0
MOVL C01904 V=800.0 PL=0
MOVL C01905 V=800.0 PL=0
MOVL C01906 V=800.0 PL=0
MOVL C01907 V=800.0 PL=0
MOVL C01908 V=800.0 PL=0
MOVL C01909 V=800.0 PL=0
MOVL C01910 V=800.0 PL=0
MOVL C01911 V=800.0 PL=0
MOVL C01912 V=800.0 PL=0
MOVL C01913 V=800.0 PL=0
MOVL C01914 V=800.0 PL=0
MOVL C01915 V=800.0 PL=0
MOVL C01916 V=800.0 PL=0
MOVL C01917 V=800.0 PL=0
MOVL C01918 V=800.0 PL=0
MOVL C01919 V=800.0 PL=0
MOVL C01920 V=800.0 PL=0
MOVL C01921 V=800.0 PL=0
MOVL C01922 V=800.0 PL=0
MOVL C01923 V=800.0 PL=0
MOVL C01924 V=800.0 PL=0
MOVL C01925 V=800.0 PL=0
MOVL C01926 V=800.0 PL=0
MOVL C01927 V=800.0 PL=0
MOVL C01928 V=800.0 PL=0
MOVL C01929 V=800.0 PL=0
MOVL C01930 V=800.0 PL=0
MOVL C01931 V=800.0 PL=0
MOVL C01932 V=800.0 PL=0
MOVL C01933 V=800.0 PL=0
MOVL C01934 V=800.0 PL=0
MOVL C01935 V=800.0 PL=0
MOVL C01936 V=800.0 PL=0
MOVL C01937 V=800.0 PL=0
MOVL C01938 V=800.0 PL=0
MOVL C01939 V=800.0 PL=0
MOVL C01940 V=800.0 PL=0
MOVL C01941 V=800.0 PL=0
MOVL C01942 V=800.0 PL=0
MOVL C01943 V=800.0 PL=0
MOVL C01944 V=800.0 PL=0
MOVL C01945 V=800.0 PL=0
MOVL C01946 V=800.0 PL=0
MOVL C01947 V=800.0 PL=0
MOVL C01948 V=800.0 PL=0
MOVL C01949 V=800.0 PL=0
MOVL C01950 V=800.0 PL=0
MOVL C01951 V=800.0 PL=0
MOVL C01952 V=800.0 PL=0
MOVL C01953 V=800.0 PL=0
MOVL C01954 V=800.0 PL=0
